# B&R Automation Studio project NAINV104C00R8L515F00 (part 30)

#### Local.var
```iecst
(*2020-09-10*)
(**)
(*Local Action, State & Status*)
VAR
	eAct : eHermesAction := HermesActIdle;
	eStat : eHermesAction := HermesActIdle;
	eMainStatus : eFBStatus := Idle;
	eStatus : eFBStatus := Idle;
	eStatus1 : eFBStatus := Idle;
	eStatus2 : eFBStatus := Idle;
	eStatus3 : eFBStatus := Idle;
	udiStatus : UDINT := 0;
	udiStatus1 : UDINT := 0;
	udiStatus2 : UDINT := 0;
	udiStatus3 : UDINT := 0;
	udiStatus4 : UDINT := 0;
	sStatTxt : STRING[200] := '';
	a_sStatText : ARRAY[0..50] OF STRING[200] := ['Idling','Background Starting Operations','Background Stopping Operations','Deleting Old Log File','Creating Directory','Writing Retain File','Reading Retain File','Saving Configuration',43('')];
END_VAR
(**)
(*Local Alarm*)
VAR
	tyAlmData : tyAlmDat;
	tyAlmData1 : tyAlmDat;
	tyAlmData2 : tyAlmDat;
	tyAlmData3 : tyAlmDat;
	tyAlmData4 : tyAlmDat;
	tyInfoData : tyAlmDat;
	a_tyAlmText : ARRAY[10000..10199] OF tyAlmTxt := [(sAlmText:='Invalid Ident While Creating Server',sRcyText:='Problem Occurred In The TCP/IP Connection. Check The Connection And Try To Reconnect.'),(sAlmText:='Setting Keep Alive Interval Time Error While Creating Server',sRcyText:='Unable To Establish Connection Between Machine. Check For Setting And Resume Operation.'),(sAlmText:='Setting Keep Alive Idle Time Error While Creating Server',sRcyText:='Unable To Establish Connection Between Machine. Check For Setting And Resume Operation.'),(sAlmText:='Setting Keep Alive Count Error While Creating Server',sRcyText:='Unable To Establish Connection Between Machine. Check For Setting And Resume Operation.'),(sAlmText:='Setting Keep Alive Error While Creating Server',sRcyText:='Unable To Establish Connection Between Machine. Check For Setting And Resume Operation.'),(sAlmText:='Setting Receive Buffer Error While Creating Server',sRcyText:='Unable To Establish Connection Between Machine. Check For Setting And Resume Operation.'),(sAlmText:='Setting Send Buffer Error While Creating Server',sRcyText:='Unable To Establish Connection Between Machine. Check For Setting And Resume Operation.'),(sAlmText:='Setting No Waiting Error While Creating Server',sRcyText:='Unable To Establish Connection Between Machine. Check For Setting And Resume Operation.'),(sAlmText:='TCP Open Port Error While Creating Server',sRcyText:='Problem Occurred In The TCP/IP Connection. Check The Connection And Try To Reconnect.'),(sAlmText:='Closing TCP Error While Creating Server',sRcyText:='Problem Occurred In The TCP/IP Connection. Check The Connection And Try To Reconnect.'),(sAlmText:='Invalid Ident While Listening Client',sRcyText:='There Was A Problem Connecting To The Server. The Server May Not Exist or It is Unavailable At This Time. Check The Connection and Try Again.'),(0),(sAlmText:='DS Hermes Connection Lost',sRcyText:='There Was A Problem Connecting To The Server. The Server May Not Exist or It is Unavailable At This Time. Check The Connection and Try Again.'),(0),(sAlmText:='Invalid Ident While Receiving Data',sRcyText:='Problem Occurred In The TCP/IP Connection. Check The Connection And Try To Reconnect.'),(sAlmText:='TCP Receive Data Error While Receiving Data',sRcyText:='Problem Occurred In The TCP/IP Connection. Check The Connection And Try To Reconnect.'),(sAlmText:='Receive BoardAvailable While Downstream In Not Connected State',sRcyText:='Receive Illegal Message.'),(sAlmText:='Receive RevokeBoardAvailable While Downstream In Not Connected State',sRcyText:='Receive Illegal Message.'),(sAlmText:='Receive MachineReady While Downstream In Not Connected State',sRcyText:='Receive Illegal Message.'),(sAlmText:='Receive RevokeMachineReady While Downstream In Not Connected State',sRcyText:='Receive Illegal Message.'),(sAlmText:='Receive StartTransport While Downstream In Not Connected State',sRcyText:='Receive Illegal Message.'),(sAlmText:='Receive StopTransport While Downstream In Not Connected State',sRcyText:='Receive Illegal Message.'),(sAlmText:='Receive TransportFinished While Downstream In Not Connected State',sRcyText:='Receive Illegal Message.'),(sAlmText:='Receive BoardForecast While Downstream In Not Connected State',sRcyText:='Receive Illegal Message.'),(sAlmText:='Receive ServiceDescription While Downstream In Service Description State',sRcyText:='Receive Illegal Message.'),(sAlmText:='Receive BoardAvailable While Downstream In Service Description State',sRcyText:='Receive Illegal Message.'),(sAlmText:='Receive RevokeBoardAvailable While Downstream In Service Description State',sRcyText:='Receive Illegal Message.'),(sAlmText:='Receive MachineReady While Downstream In Service Description State',sRcyText:='Receive Illegal Message.'),(sAlmText:='Receive RevokeMachineReady While Downstream In Service Description State',sRcyText:='Receive Illegal Message.'),(sAlmText:='Receive StartTransport While Downstream In Service Description State',sRcyText:='Receive Illegal Message.'),(sAlmText:='Receive StopTransport While Downstream In Service Description State',sRcyText:='Receive Illegal Message.'),(sAlmText:='Receive TransportFinished While Downstream In Service Description State',sRcyText:='Receive Illegal Message.'),(sAlmText:='Receive BoardForecast While Downstream In Service Description State',sRcyText:='Receive Illegal Message.'),(sAlmText:='Receive ServiceDescription While Downstream In Not Available Not Ready State',sRcyText:='Receive Illegal Message.'),(sAlmText:='Receive BoardAvailable While Downstream In Not Available Not Ready State',sRcyText:='Receive Illegal Message.'),(sAlmText:='Receive RevokeBoardAvailable While Downstream In Not Available Not Ready State',sRcyText:='Receive Illegal Message.'),(sAlmText:='Receive RevokeMachineReady While Downstream In Not Available Not Ready State',sRcyText:='Receive Illegal Message.'),(sAlmText:='Receive StartTransport While Downstream In Not Available Not Ready State',sRcyText:='Receive Illegal Message.'),(sAlmText:='Receive StopTransport While Downstream In Not Available Not Ready State',sRcyText:='Receive Illegal Message.'),(sAlmText:='Receive TransportFinished While Downstream In Not Available Not Ready State',sRcyText:='Receive Illegal Message.'),(sAlmText:='Receive BoardForecast While Downstream In Not Available Not Ready State',sRcyText:='Receive Illegal Message.'),(sAlmText:='Receive ServiceDescription While Downstream In Board Available State',sRcyText:='Receive Illegal Message.'),(sAlmText:='Receive BoardAvailable While Downstream In Board Available State',sRcyText:='Receive Illegal Message.'),(sAlmText:='Receive RevokeBoardAvailable While Downstream In Board Available State',sRcyText:='Receive Illegal Message.'),(sAlmText:='Receive RevokeMachineReady While Downstream In Board Available State',sRcyText:='Receive Illegal Message.'),(sAlmText:='Receive StartTransport While Downstream In Board Available State',sRcyText:='Receive Illegal Message.'),(sAlmText:='Receive StopTransport While Downstream In Board Available State',sRcyText:='Receive Illegal Message.'),(sAlmText:='Receive TransportFinished While Downstream In Board Available State',sRcyText:='Receive Illegal Message.'),(sAlmText:='Receive BoardForecast While Downstream In Board Available State',sRcyText:='Receive Illegal Message.'),(sAlmText:='Receive ServiceDescription While Downstream In Machine Ready State',sRcyText:='Receive Illegal Message.'),(sAlmText:='Receive BoardAvailable While Downstream In Machine Ready State',sRcyText:='Receive Illegal Message.'),(sAlmText:='Receive RevokeBoardAvailable While Downstream In Machine Ready State',sRcyText:='Receive Illegal Message.'),(sAlmText:='Receive MachineReady While Downstream In Machine Ready State',sRcyText:='Receive Illegal Message.'),(sAlmText:='Receive StopTransport While Downstream In Machine Ready State',sRcyText:='Receive Illegal Message.'),(sAlmText:='Receive TransportFinished While Downstream In Machine Ready State',sRcyText:='Receive Illegal Message.'),(sAlmText:='Receive BoardForecast While Downstream In Machine Ready State',sRcyText:='Receive Illegal Message.'),(sAlmText:='Receive ServiceDescription While Downstream In Available And Ready State',sRcyText:='Receive Illegal Message.'),(sAlmText:='Receive BoardAvailable While Downstream In Available And Ready State',sRcyText:='Receive Illegal Message.'),(sAlmText:='Receive RevokeBoardAvailable While Downstream In Available And Ready State',sRcyText:='Receive Illegal Message.'),(sAlmText:='Receive MachineReady While Downstream In Available And Ready State',sRcyText:='Receive Illegal Message.'),(sAlmText:='Receive StopTransport While Downstream In Available And Ready State',sRcyText:='Receive Illegal Message.'),(sAlmText:='Receive TransportFinished While Downstream In Available And Ready State',sRcyText:='Receive Illegal Message.'),(sAlmText:='Receive BoardForecast While Downstream In Available And Ready State',sRcyText:='Receive Illegal Message.'),(sAlmText:='Receive ServiceDescription While Downstream In Transporting State',sRcyText:='Receive Illegal Message.'),(sAlmText:='Receive BoardAvailable While Downstream In Transporting State',sRcyText:='Receive Illegal Message.'),(sAlmText:='Receive RevokeBoardAvailable While Downstream In Transporting State',sRcyText:='Receive Illegal Message.'),(sAlmText:='Receive MachineReady While Downstream In Transporting State',sRcyText:='Receive Illegal Message.'),(sAlmText:='Receive RevokeMachineReady While Downstream In Transporting State',sRcyText:='Receive Illegal Message.'),(sAlmText:='Receive StartTransport While Downstream In Transporting State',sRcyText:='Receive Illegal Message.'),(sAlmText:='Receive TransportFinished While Downstream In Transporting State',sRcyText:='Receive Illegal Message.'),(sAlmText:='Receive BoardForecast While Downstream In Transporting State',sRcyText:='Receive Illegal Message.'),(sAlmText:='Receive ServiceDescription While In Transport Finished State',sRcyText:='Receive Illegal Message.'),(sAlmText:='Receive BoardAvailable While In Transport Finished State',sRcyText:='Receive Illegal Message.'),(sAlmText:='Receive RevokeBoardAvailable While In Transport Finished State',sRcyText:='Receive Illegal Message.'),(sAlmText:='Receive MachineReady While In Transport Finished State',sRcyText:='Receive Illegal Message.'),(sAlmText:='Receive RevokeMachineReady While In Transport Finished State',sRcyText:='Receive Illegal Message.'),(sAlmText:='Receive StartTransport While In Transport Finished State',sRcyText:='Receive Illegal Message.'),(sAlmText:='Receive TransportFinished While In Transport Finished State',sRcyText:='Receive Illegal Message.'),(sAlmText:='Receive BoardForecast While In Transport Finished State',sRcyText:='Receive Illegal Message.'),(sAlmText:='Receive ServiceDescription While Downstream In Transport Stopped State',sRcyText:='Receive Illegal Message.'),(sAlmText:='Receive BoardAvailable While Downstream In Transport Stopped State',sRcyText:='Receive Illegal Message.'),(sAlmText:='Receive RevokeBoardAvailable While Downstream In Transport Stopped State',sRcyText:='Receive Illegal Message.'),(sAlmText:='Receive MachineReady While Downstream In Transport Stopped State',sRcyText:='Receive Illegal Message.'),(sAlmText:='Receive RevokeMachineReady While Downstream In Transport Stopped State',sRcyText:='Receive Illegal Message.'),(sAlmText:='Receive StartTransport While Downstream In Transport Stopped State',sRcyText:='Receive Illegal Message.'),(sAlmText:='Receive StopTransport While Downstream In Transport Stopped State',sRcyText:='Receive Illegal Message.'),(sAlmText:='LaneId Mismatch While Checking Service Description',sRcyText:='The LaneId Value Does Not Match. Change The Value And Resend The Value.'),(sAlmText:='MachineId Missing While Checking Service Description',sRcyText:='Missing Input Value For MachineId. Fill Up The Value And Resend.'),(sAlmText:='LandId Out Of Range While Checking Service Description',sRcyText:='LaneId Does Not Fall Within The Expected Range.'),(sAlmText:='LandId Missing While Checking Service Description',sRcyText:='Missing Input Value For LaneId. Fill Up The Value And Resend.'),(sAlmText:='Version Missing While Checking Service Description',sRcyText:='Missing Input Value For Version. Fill Up The Value And Resend.'),(sAlmText:='SupportedFeatures Missing While Checking Service Description',sRcyText:='Missing Input Value For SupportedFeatures. Fill Up The Value And Resend.'),(sAlmText:='NotificationCode Out Of Range While Checking Notification',sRcyText:='NotificationCode Does Not Fall Within The Expected Range.'),(sAlmText:='NotificationCode Missing While Checking Notification',sRcyText:='Missing Input Value For NotificationCode. Fill Up The Value And Resend.'),(sAlmText:='Severity Missing While Checking Notification',sRcyText:='Missing Input Value For Severity. Fill Up The Value And Resend.'),(sAlmText:='Description Missing While Checking Notification',sRcyText:='Missing Input Value For Description. Fill Up The Value And Resend.'),2((0)),(sAlmText:='FailedBoard Missing While Checking Machine Ready',sRcyText:='Missing Input Value For FailedBoard. Fill Up The Value And Resend.'),(sAlmText:='TransferState Missing While Checking Stop Transport',sRcyText:='Missing Input Value For TransferState. Fill Up The Value And Resend.'),(sAlmText:='BoardId Missing While Checking Stop Transport',sRcyText:='Missing Input Value For BoardId. Fill Up The Value And Resend.'),(sAlmText:='BoardId Missing While Checking Start Transport',sRcyText:='Missing Input Value For BoardId. Fill Up The Value And Resend.'),(sAlmText:='Barcode Missing While Checking Query Board Info',sRcyText:='Missing Input Value For BoardId. Fill Up The Value And Resend.'),(0),(sAlmText:='BoardId Mismatch While Checking Start Transport & Stop Transport',sRcyText:='The BoardId Value Does Not Match. Change The Value And Resend The Value.'),(sAlmText:='BoardId Missing While Checking Start Transport & Stop Transport',sRcyText:='Missing Input Value For BoardId. Fill Up The Value And Resend.'),(sAlmText:='Service Description Interchange Time Out',sRcyText:='Timeout Expired Before Operation Completed. Reset And Resume Operation.'),(sAlmText:='Transport Time Out',sRcyText:='Timeout Expired Before Operation Completed. Reset And Resume Operation.'),(sAlmText:='Receive TransportFinished While Downstream In Transport Stopped State',sRcyText:='Receive Illegal Message.'),(sAlmText:='Receive BoardForecast While Downstream In Transport Stopped State',sRcyText:='Receive Illegal Message.'),(sAlmText:='Stop Transport Request To Send From Upstream Hermes',sRcyText:='Sending Illegal Message.'),(sAlmText:='Get Directory Info Error While Deleting Old Log',sRcyText:='An Error Was Encountered While Getting Directory Info. Please Contact Nutek For A Possible Solution.'),(sAlmText:='Directory Read Error While Deleting Old Log',sRcyText:='An Error Was Encountered While Reading Directory. Please Contact Nutek For A Possible Solution.'),(sAlmText:='File Delete Error While Deleting Old Log',sRcyText:='An Error Was Encountered While Trying To Delete File. Please Contact Nutek For A Possible Solution.'),18((0)),(sAlmText:='Check Alive Time Out',sRcyText:='Timeout Expired Before Operation Completed. Reset And Resume Operation.'),(sAlmText:='Waiting Check Alive Time Out',sRcyText:='Timeout Expired Before Operation Completed. Reset And Resume Operation.'),(sAlmText:='Check Alive Id Mismatch',sRcyText:='The Check Alive Id Value Does Not Match. Change The Value And Resend The Value.'),(sAlmText:='Machine Ready Request To Send From Upstream Hermes',sRcyText:='Sending Illegal Message.'),(sAlmText:='Revoke Machine Ready Request To Send From Upstream Hermes',sRcyText:='Sending Illegal Message.'),(sAlmText:='Start Transport Request To Send From Upstream Hermes',sRcyText:='Sending Illegal Message.'),(sAlmText:='Set Configuration Request To Send From Upstream Hermes',sRcyText:='Sending Illegal Message.'),(sAlmText:='Get Configuration Request To Send From Upstream Hermes',sRcyText:='Sending Illegal Message.'),(sAlmText:='Current Configuration Request To Send From Upstream Hermes',sRcyText:='Sending Illegal Message.'),(sAlmText:='Board Forecast Request To Send From Upstream Hermes',sRcyText:='Sending Illegal Message.'),(sAlmText:='Query Board Info Request To Send From Upstream Hermes',sRcyText:='Sending Illegal Message.'),(sAlmText:='Invalid Ident While Sending Data',sRcyText:='Invalid Ident Value.'),(sAlmText:='TCP Retry Send Data Error While Sending Data',sRcyText:='Problem Occurred In The TCP/IP Connection. Check The Connection And Try To Reconnect.'),(sAlmText:='TCP Send Data Error',sRcyText:='Problem Occurred In The TCP/IP Connection. Check The Connection And Try To Reconnect.'),(sAlmText:='Invalid Ident While Closing TCP',sRcyText:='Invalid Ident Value.'),(sAlmText:='Closing TCP Error',sRcyText:='Problem Occurred In The TCP/IP Connection. Check The Connection And Try To Reconnect.'),(sAlmText:='File Open Error While Writing Log',sRcyText:='An Error Was Encountered While Trying To Open File. Please Contact Nutek For A Possible Solution.'),(sAlmText:='File Create Error While Writing Log',sRcyText:='An Error Was Encountered While Trying To Create File. Please Contact Nutek For A Possible Solution.'),(sAlmText:='Get File Info Error While Writing Log',sRcyText:='An Error Was Encountered While Getting File Info. Please Contact Nutek For A Possible Solution.'),(sAlmText:='File Write Error While Writing Log',sRcyText:='An Error Was Encountered While Trying To Write File. Please Contact Nutek For A Possible Solution.'),(sAlmText:='File Close Error While Writing Log',sRcyText:='An Error Was Encountered While Trying To Close File. Please Contact Nutek For A Possible Solution.'),(sAlmText:='Directory Does Not Exist While Writing Log',sRcyText:='The Directory Does Not Exist.Please Contact Nutek For A Possible Solution.'),(sAlmText:='Invalid Ident While Closing TCP',sRcyText:='Invalid Ident Value.'),(sAlmText:='Closing TCP Error',sRcyText:='Problem Occurred In The TCP/IP Connection. Check The Connection And Try To Reconnect.'),(0),(sAlmText:='Board Jam At Sensor After Transfer Interrupted',sRcyText:='Pull Back Board From Downstream Machine'),42((0))];
END_VAR
(**)
(*Local Output*)
VAR
	bConnected : BOOL;
	bHandshakeDone : BOOL;
	bUSRdy : BOOL;
	bDSRdy : BOOL;
	bUSGdRdy : BOOL;
	bDSGdRdy : BOOL;
	bTransporting : BOOL;
	bStopTransport : BOOL;
	sInternalSnd : STRING[65535];
END_VAR
(**)
(*Local Input*)
VAR
	udiRstErr : UDINT := 0;
	bPrep : BOOL := TRUE;
	bEn : BOOL := TRUE;
	bDis : BOOL := FALSE;
	tyParam : tyHermesDSParam;
	sIPAddr : STRING[15] := '192.168.0.100';
	a_usiMacAddr : ARRAY[0..5] OF USINT := [6(0)];
	tyDTStructure : DTStructure := (year:=2019,month:=01,day:=05,wday:=05,hour:=21,minute:=28,second:=30,millisec:=123,microsec:=456);
	dtCurrDT : DATE_AND_TIME := DT#2019-02-23-12:30:50;
	bRdySnd : BOOL := FALSE;
	bSndCompl : BOOL := FALSE;
	bSndInCompl : BOOL := FALSE;
	bSndNotStart : BOOL := FALSE;
	bBAWidthEn : BOOL := TRUE; (*Board Available Check Width*)
	bBASltEn : BOOL := FALSE; (*Board Available Check Slot*)
	bBFWidthEn : BOOL := TRUE; (*Board Available Check Width*)
	bBFSltEn : BOOL := FALSE; (*Board Available Check Slot*)
	sMcId : STRING[80] := '';
	sInterfaceId : STRING[80];
	sVersion : STRING[7] := '1.0.2';
	eFailedBoard : eHermesFailedBoard := HermesUnknownBoard;
	sRecipeNm : STRING[254] := '';
	eFlippedBoard : eHermesFlippedBoard := HermesFlippedBoardUnknownSide;
	sTopBarcode : STRING[254] := '';
	sBottomBarcode : STRING[254] := '';
	rLength : REAL := 0;
	rThickness : REAL := 0;
	rConveyorSpeed : REAL := 0;
	rTopClearanceHeight : REAL := 0;
	rBottomClearanceHeight : REAL := 0;
	rWeight : REAL := 0;
	sWorkOrderId : STRING[80] := '';
	sBatchId : STRING[80] := '';
	diWidthInUM : DINT := 0;
	diMinSltValue : DINT := 0;
	diMaxSltValue : DINT := 0;
	diPitch : DINT := 0;
	diTtlSlt : DINT := 0;
	diSltToSltInUM : DINT := 0;
	udiSndBffrSize : UDINT := 65536;
	udiRcvBffrSize : UDINT := 65536;
	udiAliveIdleTimeInSec : UDINT := 5;
	tConnTimeOut : TIME := T#30s;
	diTransferInTO : DINT := 30000;
	a_tyXMLTableDataBrdAvl : ARRAY[0..200] OF tyXMLTableDat;
	iXMLTableDataBrdAvlTtlIdx : INT := 0;
	bNewBrdAvl : BOOL := FALSE;
	bOpsRun : BOOL := FALSE;
	bInterruptSen : BOOL := FALSE;
	udiFileKeepDay : UDINT := 30;
	sProgNm : STRING[15] := 'DSHermes';
	bNtSettingsLoadDone : BOOL := TRUE;
	sRmtMcId : STRING[80];
	bRmtPrep : BOOL := FALSE;
	bRmtEn : BOOL := FALSE;
	bInternalUse : BOOL;
	sInternalRcv : STRING[65535];
END_VAR
(**)
(*Local*)
VAR
	bRstErr : BOOL;
	udiRstErrOld : UDINT;
	bInitDone : BOOL;
	bInitialDone : BOOL;
	bRun : BOOL;
	bStop : BOOL;
	bRstConnection : BOOL;
	bRstState : BOOL;
	udiSvrIdent : UDINT;
	udiClntIdent : UDINT;
	udiClntIdentExtra : UDINT;
	udiXMLTableWriteIdx : UDINT;
	udiMsgSendBffr : UDINT;
	udiMsgCmdBffr : UDINT;
	udiSndMsgLen : UDINT;
	sSnd : STRING[65535];
	sRcv : STRING[65535];
	a_tyXMLTableDataRcv : ARRAY[0..200] OF tyXMLTableDat;
	a_tyXMLTableDataSnd : ARRAY[0..200] OF tyXMLTableDat;
	a_eMsgSend : ARRAY[0..50] OF eHermesMsgType;
	a_eCommandSndQ : ARRAY[0..20] OF eHermesCommand;
	tyMsgTypeRcv : tyHermesMsgType;
	tyCheckAliveSnd : tyHermesCheckAlive;
	tyCheckAlivePingSnd : tyHermesCheckAlive;
	tyCheckAlivePongSnd : tyHermesCheckAlive;
	tyCheckAliveRcv : tyHermesCheckAlive;
	tyCheckAlivePingRcv : tyHermesCheckAlive;
	tyCheckAlivePongRcv : tyHermesCheckAlive;
	tyServiceDescriptionSnd : tyHermesServiceDescription;
	tyServiceDescriptionRcv : tyHermesServiceDescription;
	tyNotificationSnd : tyHermesNotification;
	tyNotificationRcv : tyHermesNotification;
	tyBoardAvailableRcv : tyHermesBoardAvailable;
	tyBoardAvailableSnd : tyHermesBoardAvailable;
	a_tyBoardDepartedInfo : ARRAY[0..49] OF tyHermesBoardAvailable;
	a_tyBoardDepartedInfoWr : ARRAY[0..49] OF tyHermesBoardAvailable;
	tyMachineReady : tyHermesMachineReady;
	tyStartTransport : tyHermesStartTransport;
	tyStopTransport : tyHermesStopTransport;
	tyTransportFinished : tyHermesTransportFinished;
	tySetConfiguration : tyHermesSetConfiguration;
	tyCurrentConfiguration : tyHermesCurrentConfiguration;
	tyBoardForecastRcv : tyHermesBoardForecast;
	tyBoardForecastSnd : tyHermesBoardForecast;
	tyQueryBoardInfo : tyHermesQueryBoardInfo;
	tySendBoardInfo : tyHermesSendBoardInfo;
	tyCommandRcv : tyHermesCommand;
	tyCommandSnd : tyHermesCommand;
	fbCreateSvr : fbTCPCreateSvr;
	fbListen : fbTCPListen;
	fbRcv : fbTCPRcv;
	fbSend : fbTCPSnd;
	fbCloseSvr : fbTCPClose;
	fbCloseClnt : fbTCPClose;
	fbParseXMLTable : fbHermesParseXMLTable;
	fbParseBrdAvlExternal : fbHermesParseXMLTable;
	fbCheckAlive : fbHermesCheckAlive;
	fbCheckAliveSendPing : fbHermesCheckAliveSendPing;
	fbCheckAliveRcvPing : fbHermesCheckAliveRcvPing;
	fbSequenceDS : fbHermesSequenceDS;
	fbSequenceTO : fbHermesSequenceTO;
END_VAR
VAR RETAIN
	usiBAIndex : USINT := 0;
END_VAR
VAR
	usiPrevBAIndex : USINT;
	eStatOld : eHermesAction := HermesActIdle;
	tyParamOld : tyHermesDSParam;
	udiLogCntr : UDINT := 1;
	udiWriteLogCntr : UDINT := 1;
	a_sLogList : ARRAY[1..10] OF STRING[65535];
	sDT : STRING[80];
	dtCurrDTTemp : DATE_AND_TIME;
	fbFileAppend1 : fbFileFullAppend;
	fbFileOldDel1 : fbFileOldDel;
	fbFileRead1 : fbFileFullRead;
	fbFileWrite1 : fbFileFullWrite;
	iWriteLogStep : INT := 0;
	tyUSHermestyBoardAvailable : tyHermesBoardAvailable;
	tyCommandParam : tyHermesCommandParam;
	bDummy : BOOL;
	bFeatureBoardForecast : BOOL;
	bNewProduct : BOOL;
	bNewWidth : BOOL;
	bNewChangeOver : BOOL;
	tySendBoardInfoAcc : tyHermesSendBoardInfo;
	rMachineCycleTime : REAL;
	rAWCycleTm : REAL;
	bFileNotFound : BOOL;
	bSendBFId : BOOL;
	bBFIdSent : BOOL;
	bSendBFNoID : BOOL;
	bSndReverseBF : BOOL;
	bRstSendBFId : BOOL;
	bFirstZoneHaveBoard : BOOL;
	bFirstZoneEndSen : BOOL;
	bAllZoneEmpty : BOOL;
	bTransportFinishedSnd : BOOL;
	fbTimerRstBFId : TON;
	sInfoMcRdyMsg : STRING[200];
	sTempRealWidth : STRING[15];
	sRstTim : STRING[15];
	udiModuleNum : UDINT := 3351;
END_VAR
(*Send Board Info*)
VAR
	bSearchTop : BOOL;
	bSearchBottom : BOOL;
	siTopBarcodeIdx : SINT;
	siBottomBarcodeIdx : SINT;
	siSearhIdx : SINT;
	siFoundIdx : SINT;
	bCompleteSearch : BOOL;
END_VAR
(*Route*)
VAR
	bTriggerRouteReversal : BOOL;
	bReverseDSSndBfWBrdID : BOOL;
	bSwitchtoReverseSend : BOOL;
	fbRstReverseSndGate : TON;
	bNotifyRstReverseSndGate : BOOL;
	bBlkDS : BOOL;
	bProcessRouteEn : BOOL;
	bManualRmvRoute : BOOL;
	bReturnRoute : BOOL;
	bNomRouteEn : BOOL;
	bReverseSentRoute : BOOL;
	usiUSHermesReverseDSSendBFId : USINT;
	bUSHermesProcessRouteTrigger : BOOL;
	iRoute : INT;
	iAction : INT;
	bDSHermesRcvReverseUSMcRdy : BOOL;
	bReverseRcvBlkDS : BOOL;
END_VAR
```

#### Act_Action.st
```iecst
(** 2021-08-01 **)
ACTION Act_Action:

	//Reset Error
	IF (eStatus = Error) AND bRstErr THEN
		p_eAct	:= HermesActIdle;
		eStat	:= HermesActIdle;
	END_IF

	//Set p_eAct
	IF eStatus = Idle  OR eStatus = Done THEN //OR eStatus = Busy
		eStat	:= p_eAct;
	END_IF

END_ACTION
```

#### Act_Alarm.st
```iecst
(** 2021-08-01 **)
ACTION Act_Alarm:

	//Error
	IF EDGEPOS(eStatus = Error) THEN

		tyAlmData.sProgNm		:= p_sProgNm;
		tyAlmData.udiCode		:= udiStatus;
		tyAlmData.eSeverity		:= AlmSeverityError;
		tyAlmData.udiRunTime	:= tyAlmData.udiRunTime + 1;
		tyAlmData.bAlm			:= TRUE;
		tyAlmData.udiModuleNum  := udiModuleNum;
		g_sDSHermesProgNm		:= p_sProgNm;

		//Get Error Message
		IF tyAlmData.udiCode < 10000 OR tyAlmData.udiCode > 10199 THEN
			tyAlmData.sAlmMsg	:= 'Unknown';
			tyAlmData.sRcyMsg	:= 'Unknown';
		ELSE
			tyAlmData.sAlmMsg	:= a_tyAlmText[tyAlmData.udiCode].sAlmText;
			tyAlmData.sRcyMsg	:= a_tyAlmText[tyAlmData.udiCode].sRcyText;
		END_IF

		sStatTxt	:= tyAlmData.sAlmMsg;

	ELSIF bRstErr AND (tyAlmData.udiCode <> 0) THEN

		tyAlmData.udiCode	:= 0;
		tyAlmData.eSeverity	:= AlmSeverityNA;
		tyAlmData.sAlmMsg	:= '';
		tyAlmData.sRcyMsg	:= '';
		tyAlmData.bAlm			:= FALSE;
		sStatTxt	:= a_sStatText[eStat];

	END_IF

END_ACTION
```

#### Act_Alarm1.st
```iecst
(** 2021-08-01 **)
ACTION Act_Alarm1: //General

	//Error
	IF EDGEPOS(eStatus1 = Error) THEN

		tyAlmData1.sProgNm		:= p_sProgNm;
		tyAlmData1.udiCode		:= udiStatus1;
		tyAlmData1.eSeverity	:= AlmSeverityError;
		tyAlmData1.udiRunTime	:= tyAlmData1.udiRunTime + 1;
		tyAlmData1.bAlm			:= TRUE;
		tyAlmData1.udiModuleNum := udiModuleNum;
		g_sDSHermesProgNm		:= p_sProgNm;

		//Get Error Message
		IF tyAlmData1.udiCode < 10000 OR tyAlmData1.udiCode > 10199 THEN
			tyAlmData1.sAlmMsg	:= 'Unknown';
			tyAlmData1.sRcyMsg	:= 'Unknown';
		ELSE
			tyAlmData1.sAlmMsg	:= a_tyAlmText[tyAlmData1.udiCode].sAlmText;
			tyAlmData1.sRcyMsg	:= a_tyAlmText[tyAlmData1.udiCode].sRcyText;
		END_IF

		sStatTxt	:= tyAlmData1.sAlmMsg;

	ELSIF bRstErr AND (tyAlmData1.udiCode <> 0) THEN

		tyAlmData1.udiCode		:= 0;
		tyAlmData1.eSeverity	:= AlmSeverityNA;
		tyAlmData1.sAlmMsg		:= '';
		tyAlmData1.sRcyMsg		:= '';
		tyAlmData1.bAlm			:= FALSE;
		sStatTxt	:= a_sStatText[eStat];

	END_IF

END_ACTION
```

#### Act_Background_BoardForecast.st
```iecst
(** 2023-08-01 **)
ACTION Act_Background_BoardForecast:

//	bSndReverseBF := p_bUSHermesReverseDSSendBFId

	bFeatureBoardForecast := (p_tyParam.bFeatureBoardForecast = TRUE) AND (tyServiceDescriptionRcv.tyAvl.tySupportedFeatures.bFeatureBoardForecast = TRUE) (*AND bHandshakeDone*) ;

	IF NOT(bFeatureBoardForecast) THEN
		bNewChangeOver := FALSE;
		bSendBFNoID	   := FALSE;
		bSendBFId	   := FALSE;
		bBFIdSent	   := FALSE;
		bSndReverseBF  :=  FALSE;
		tyInfoData.sProgNm		:= '';
		tyInfoData.udiCode		:= 0;
		tyInfoData.eSeverity	:= AlmSeverityNA;
		tyInfoData.sAlmMsg		:= '';
	ELSE
		bSndReverseBF := EDGEPOS(p_usiUSHermesReverseDSSendBFId <> 0);

		fbTimerRstBFId(IN:= bSendBFId AND bBFIdSent
		AND NOT(bRstSendBFId) AND tyInfoData.udiCode= 10999
		AND bDSRdy
		,PT := T#1000s); //start counting when received mismatch Machine ready

		IF bRstSendBFId OR fbTimerRstBFId.Q
			OR EDGEPOS(bAllZoneEmpty AND p_bConvInitDone)  THEN //Reset BoardForecast width id
			bRstSendBFId := FALSE;
			bSendBFId := FALSE;
			bBFIdSent := FALSE;
		ELSIF fbTimerRstBFId.IN THEN
			sRstTim 				:= REAL_TO_STRING(TIME_TO_REAL(fbTimerRstBFId.PT-fbTimerRstBFId.ET)/1000.0);
			tyInfoData.sAlmMsg		:= CONCAT(sInfoMcRdyMsg,CONCAT(sRstTim,'(seconds)'));
		END_IF

		IF EDGEPOS(bNewProduct) OR EDGEPOS(bNewWidth) THEN  //Trigger BFID
			bNewChangeOver := TRUE;
			bBFIdSent := FALSE; //To resend BF-ID
		END_IF

		IF bNewChangeOver AND bAllZoneEmpty AND p_bConvInitDone THEN
			bNewChangeOver:= FALSE;
			bSendBFId	  := TRUE; //reset when find mactch machine ready
		END_IF

		IF bSendBFId = FALSE AND bBFIdSent = FALSE THEN //reset notification
			tyInfoData.sProgNm		:= '';
			tyInfoData.udiCode		:= 0;
			tyInfoData.eSeverity	:= AlmSeverityNA;
			tyInfoData.sAlmMsg		:= '';
		END_IF

		IF bSendBFId = FALSE   THEN  	//Trigger BF No Id
			bSendBFNoID	:= FALSE;
			IF bFirstZoneHaveBoard AND NOT(bFirstZoneEndSen) THEN //Zone 1 PCB_In and have Board
				bSendBFNoID	:= TRUE;
			ELSIF bSndReverseBF THEN//EDGEPOS(bSndReverseBF) OR EDGENEG(bSndReverseBF) THEN //Reverse route
				bSendBFNoID	:= TRUE; //EDGEPOS send Brd id , EDGENEG send empty brd id
			END_IF
		END_IF

	END_IF

END_ACTION
```

#### Act_Background_ChgConfig.st
```iecst
(** 2021-08-01 **)
ACTION Act_Background_ChgConfig:

	IF eStatus2 <> Error THEN

		IF (tyParamOld.iLaneID <> p_tyParam.iLaneID) OR (tyParamOld.sClientAddress <> p_tyParam.sClientAddress) OR (tyParamOld.uiClientPort <> p_tyParam.uiClientPort) OR (tyParamOld.uiSvrPort <> p_tyParam.uiSvrPort)
			OR (tyParamOld.bFeatureBoardForecast <> p_tyParam.bFeatureBoardForecast) OR (tyParamOld.bFeatureCheckAliveResponse <> p_tyParam.bFeatureCheckAliveResponse) OR (tyParamOld.bFeatureSendBoardInfo <> p_tyParam.bFeatureSendBoardInfo) THEN

			IF udiClntIdent <> 0 THEN
				fHermesAddOneMsgSend(ADR(a_eMsgSend) , ADR(udiMsgSendBffr) , HermesMsgTypeNotification);

				tyNotificationSnd.tyAvl.bSeverity			:= TRUE;
				tyNotificationSnd.tyAvl.bNotificationCode	:= TRUE;
				tyNotificationSnd.tyAvl.bDescription		:= TRUE;
				tyNotificationSnd.tyData.eSeverity			:= HermesSeverityFatalError;
				tyNotificationSnd.tyData.iNotificationCode	:= 3;
				tyNotificationSnd.tyData.sDescription		:= 'Configuration Changed';

			END_IF

			bRstConnection	:= TRUE;

		END_IF

	END_IF

END_ACTION
```

#### Act_Background_ChkAlive.st
```iecst
(** 2019-05-30 **)
ACTION Act_Background_ChkAlive:

	IF eStatus1 <> Error THEN

		//Standard Check Alive (Without Ping & Pong)
		fbCheckAlive.bDataRcv		:= tyMsgTypeRcv.bCheckAlive OR tyMsgTypeRcv.bMachineReady OR tyMsgTypeRcv.bRevokeMachineReady OR tyMsgTypeRcv.bStartTransport OR tyMsgTypeRcv.bStopTransport OR tyMsgTypeRcv.bQueryBoardInfo;
		fbCheckAlive.tSendTm		:= p_tyParam.tSndAlive;
		fbCheckAlive.tRcvTimeOut	:= p_tyParam.tRcvAlive;
		fbCheckAlive(bEn := TRUE);

		IF fbCheckAlive.udiStatus > 0 AND fbCheckAlive.udiStatus < 65534 THEN
			eStatus1	:= Error;

			IF fbCheckAlive.udiStatus = 2767 THEN
				udiStatus1	:= 10132;	//Check Alive Time Out
			ELSE
				udiStatus1	:= fbCheckAlive.udiStatus;
			END_IF

			fHermesAddOneMsgSend(ADR(a_eMsgSend) , ADR(udiMsgSendBffr) , HermesMsgTypeNotification);

			tyNotificationSnd.tyAvl.bSeverity			:= TRUE;
			tyNotificationSnd.tyAvl.bNotificationCode	:= TRUE;
			tyNotificationSnd.tyAvl.bDescription		:= TRUE;
			tyNotificationSnd.tyData.eSeverity			:= HermesSeverityFatalError;
			tyNotificationSnd.tyData.iNotificationCode	:= UDINT_TO_INT(udiStatus1);
			tyNotificationSnd.tyData.sDescription		:= a_tyAlmText[udiStatus1].sAlmText;

		ELSE
			IF EDGEPOS(fbCheckAlive.bDataSend) THEN
				fHermesAddOneMsgSend(ADR(a_eMsgSend) , ADR(udiMsgSendBffr) , HermesMsgTypeCheckAlive);
				tyCheckAliveSnd	:= fbCheckAlive.tyDataSend;
			END_IF

		END_IF

		tyMsgTypeRcv.bCheckAlive	:= FALSE;	//Reset Check Alive

	END_IF

END_ACTION
```

#### Act_Background_CmpParamRcv.st
```iecst
(** 2021-08-01 **)
ACTION Act_Background_CmpParamRcv:

	IF eStatus2 <> Error THEN

		IF tyMsgTypeRcv.bStopTransport = TRUE THEN
			udiStatus2	:= fHermesChkParamSTST(tyStartTransport , tyStopTransport);

			IF udiStatus2 <> 0 THEN
				eStatus2	:= Error;

				IF udiStatus2 = 2712 THEN
					udiStatus2	:= 10104;	//BoardId Mismatch While Checking Start Transport & Stop Transport
				ELSIF udiStatus2 = 2713 THEN
					udiStatus2	:= 10105;	//BoardId Missing While Checking Start Transport & Stop Transport
				END_IF

				fHermesAddOneMsgSend(ADR(a_eMsgSend) , ADR(udiMsgSendBffr) , HermesMsgTypeNotification);

				tyNotificationSnd.tyAvl.bSeverity			:= TRUE;
				tyNotificationSnd.tyAvl.bNotificationCode	:= TRUE;
				tyNotificationSnd.tyAvl.bDescription		:= TRUE;
				tyNotificationSnd.tyData.eSeverity			:= HermesSeverityFatalError;
				tyNotificationSnd.tyData.iNotificationCode	:= UDINT_TO_INT(udiStatus2);
				tyNotificationSnd.tyData.sDescription		:= a_tyAlmText[udiStatus2].sAlmText;

			END_IF
		END_IF

		IF tyMsgTypeRcv.bStartTransport = TRUE THEN
			IF fHermesChkParamBAST(tyBoardAvailableSnd , tyStartTransport) <> 0 THEN
				p_bSndNotStart	:= TRUE;
			END_IF
		END_IF

		IF bFeatureBoardForecast THEN	//HermesMsgTypeBoardForecast
			IF fbSequenceDS.eState = HermesStateMachineReady   AND bSendBFId AND bBFIdSent THEN
				udiStatus2	:= fHermesChkParamBFMR(tyBoardForecastSnd , tyMachineReady); //Modify this if our machine need to Error when ForecastId in MachineReady(Id) received is different

				IF udiStatus2 <> 0 THEN //Alarm Info
					memset(ADR(sInfoMcRdyMsg),0,SIZEOF(sInfoMcRdyMsg));
					sInfoMcRdyMsg := CONCAT(sInfoMcRdyMsg , 'Details mismatch between BoardForecast and MachineReady');
					sInfoMcRdyMsg := CONCAT(sInfoMcRdyMsg , '$r$n');
					IF udiStatus2 = 2716 THEN 	//Forecast Id Mismatch While Checking BoardForecast & Machine Ready
						sInfoMcRdyMsg := CONCAT(sInfoMcRdyMsg , 'ForecastID sent:');
						sInfoMcRdyMsg := CONCAT(sInfoMcRdyMsg , tyBoardForecastSnd.tyData.sForecastId);
						sInfoMcRdyMsg := CONCAT(sInfoMcRdyMsg , '$r$n');
						sInfoMcRdyMsg := CONCAT(sInfoMcRdyMsg , 'ForecastID received:');
						sInfoMcRdyMsg := CONCAT(sInfoMcRdyMsg , tyMachineReady.tyData.sForecastId);
					ELSIF udiStatus2 = 2717 THEN 	//Product Type Id Mismatch While Checking BoardForecast & Machine Ready
						sInfoMcRdyMsg := CONCAT(sInfoMcRdyMsg , 'ProductType sent:');
						sInfoMcRdyMsg := CONCAT(sInfoMcRdyMsg , tyBoardForecastSnd.tyData.sProductTypeId);
						sInfoMcRdyMsg := CONCAT(sInfoMcRdyMsg , '$r$n');
						sInfoMcRdyMsg := CONCAT(sInfoMcRdyMsg , 'ProductType received:');
						sInfoMcRdyMsg := CONCAT(sInfoMcRdyMsg , tyMachineReady.tyData.sProductTypeId);
					ELSIF udiStatus2 = 2718 THEN //Width Mismatch While Checking Board Forecast & Machine Ready
						sInfoMcRdyMsg := CONCAT(sInfoMcRdyMsg , 'Width sent:');
						sTempRealWidth := REAL_TO_STRING(tyBoardForecastSnd.tyData.rWidth);
						sInfoMcRdyMsg := CONCAT(sInfoMcRdyMsg ,sTempRealWidth );
						sInfoMcRdyMsg := CONCAT(sInfoMcRdyMsg , '$r$n');
						sInfoMcRdyMsg := CONCAT(sInfoMcRdyMsg , 'Width received:');
						sTempRealWidth := REAL_TO_STRING(tyMachineReady.tyData.rWidth);
						sInfoMcRdyMsg := CONCAT(sInfoMcRdyMsg , sTempRealWidth);
					END_IF
					sInfoMcRdyMsg := CONCAT(sInfoMcRdyMsg , '$r$n');
					sInfoMcRdyMsg := CONCAT(sInfoMcRdyMsg , 'Waiting New MachineReady or Ignore in:');

					tyInfoData.sProgNm		:= p_sProgNm;
					tyInfoData.udiCode		:= 10999;
					tyInfoData.eSeverity	:= AlmSeverityInfo;
					tyInfoData.sAlmMsg		:= sInfoMcRdyMsg;

				ELSE
					bRstSendBFId := TRUE; //Reset bSendBFId if MachineReady(Id) or MachineReady() received is ok
				END_IF

			END_IF
		END_IF

	END_IF

END_ACTION
```

#### Act_Background_Command.st
```iecst
(** 2021-08-01 **)
ACTION Act_Background_Command:
	//tyServiceDescriptionRcv.tyAvl.tySupportedFeatures.bFeatureCommand = TRUE AND p_tyParam.bFeatureCommand AND

	IF NOT(p_tyParam.bFeatureCommand AND tyServiceDescriptionRcv.tyAvl.tySupportedFeatures.bFeatureCommand AND bHandshakeDone) THEN
		IF tyCommandParam.a_eCommandSndQ[0] <> HermesCommandUndefined THEN
			fHermesRmvOneCmdTyp(ADR(tyCommandParam.a_eCommandSndQ),ADR(tyCommandParam.udiMsgCmdBffr));
		END_IF
	ELSE
		IF eStatus2 <> Error THEN
			//receive command

			IF tyMsgTypeRcv.bCommand THEN
				tyCommandParam.usiCommandIdx :=  tyCommandParam.usiCommandIdx + 1;
				tyCommandParam.eCommand := tyCommandRcv.tyData.eCommand;
				tyMsgTypeRcv.bCommand  := FALSE;
			END_IF

			//sending
			IF  tyCommandParam.a_eCommandSndQ[0] <> HermesCommandUndefined THEN
				//Queuing for sending command
				fHermesAddOneMsgSend(ADR(a_eMsgSend) , ADR(udiMsgSendBffr) , HermesMsgTypeCommand);
				tyCommandSnd.tyData.eCommand :=  tyCommandParam.a_eCommandSndQ[0];
				tyCommandSnd.tyAvl.bCommand :=  TRUE;
				fHermesRmvOneCmdTyp(ADR(tyCommandParam.a_eCommandSndQ),ADR(tyCommandParam.udiMsgCmdBffr));
			END_IF
		END_IF
	END_IF

END_ACTION
```

#### Act_Background_Err.st
```iecst
(** 2021-08-01 **)
ACTION Act_Background_Err:

	IF bTransporting = TRUE THEN
		IF bStopTransport AND p_bInterruptSen THEN
			eStatus2	:= Error;
			udiStatus2	:= 10157;	//Board Jam At Sensor After Transfer Interrupted
		END_IF
	END_IF

END_ACTION
```

#### Act_Background_IllegalMsg.st
```iecst
(** 2021-08-01 **)
ACTION Act_Background_IllegalMsg:

	IF eStatus2 <> Error THEN

		udiStatus2	:= fHermesIllegalMsgDS(fbSequenceDS.eState , tyMsgTypeRcv);

		IF udiStatus2 <> 0 THEN
			eStatus2	:= Error;

			IF udiStatus2 = 2840 THEN
				udiStatus2	:= 10016;	//Receive BoardAvailable While Downstream In Not Connected State
			ELSIF udiStatus2 = 2841 THEN
				udiStatus2	:= 10017;	//Receive RevokeBoardAvailable While Downstream In Not Connected State
			ELSIF udiStatus2 = 2842 THEN
				udiStatus2	:= 10018;	//Receive MachineReady While Downstream In Not Connected State
			ELSIF udiStatus2 = 2843 THEN
				udiStatus2	:= 10019;	//Receive RevokeMachineReady While Downstream In Not Connected State
			ELSIF udiStatus2 = 2844 THEN
				udiStatus2	:= 10020;	//Receive StartTransport While Downstream In Not Connected State
			ELSIF udiStatus2 = 2845 THEN
				udiStatus2	:= 10021;	//Receive StopTransport While Downstream In Not Connected State
			ELSIF udiStatus2 = 2846 THEN
				udiStatus2	:= 10022;	//Receive TransportFinished While Downstream In Not Connected State
			ELSIF udiStatus2 = 2847 THEN
				udiStatus2	:= 10023;	//Receive BoardForecast While Downstream In Not Connected State
			ELSIF udiStatus2 = 2848 THEN
				udiStatus2	:= 10024;	//Receive ServiceDescription While Downstream In Service Description State
			ELSIF udiStatus2 = 2849 THEN
				udiStatus2	:= 10025;	//Receive BoardAvailable While Downstream In Service Description State
			ELSIF udiStatus2 = 2850 THEN
				udiStatus2	:= 10026;	//Receive RevokeBoardAvailable While Downstream In Service Description State
			ELSIF udiStatus2 = 2851 THEN
				udiStatus2	:= 10027;	//Receive MachineReady While Downstream In Service Description State
			ELSIF udiStatus2 = 2852 THEN
				udiStatus2	:= 10028;	//Receive RevokeMachineReady While Downstream In Service Description State
			ELSIF udiStatus2 = 2853 THEN
				udiStatus2	:= 10029;	//Receive StartTransport While Downstream In Service Description State
			ELSIF udiStatus2 = 2854 THEN
				udiStatus2	:= 10030;	//Receive StopTransport While Downstream In Service Description State
			ELSIF udiStatus2 = 2855 THEN
				udiStatus2	:= 10031;	//Receive TransportFinished While Downstream In Service Description State
			ELSIF udiStatus2 = 2856 THEN
				udiStatus2	:= 10032;	//Receive BoardForecast While Downstream In Service Description State
			ELSIF udiStatus2 = 2857 THEN
				udiStatus2	:= 10033;	//Receive ServiceDescription While Downstream In Not Available Not Ready State
			ELSIF udiStatus2 = 2858 THEN
				udiStatus2	:= 10034;	//Receive BoardAvailable While Downstream In Not Available Not Ready State
			ELSIF udiStatus2 = 2859 THEN
				udiStatus2	:= 10035;	//Receive RevokeBoardAvailable While Downstream In Not Available Not Ready State
			ELSIF udiStatus2 = 2860 THEN
				udiStatus2	:= 10036;	//Receive RevokeMachineReady While Downstream In Not Available Not Ready State
			ELSIF udiStatus2 = 2861 THEN
				udiStatus2	:= 10037;	//Receive StartTransport While Downstream In Not Available Not Ready State
			ELSIF udiStatus2 = 2862 THEN
				udiStatus2	:= 10038;	//Receive StopTransport While Downstream In Not Available Not Ready State
			ELSIF udiStatus2 = 2863 THEN
				udiStatus2	:= 10039;	//Receive TransportFinished While Downstream In Not Available Not Ready State
			ELSIF udiStatus2 = 2864 THEN
				udiStatus2	:= 10040;	//Receive BoardForecast While Downstream In Not Available Not Ready State
			ELSIF udiStatus2 = 2865 THEN
				udiStatus2	:= 10041;	//Receive ServiceDescription While Downstream In Board Available State
			ELSIF udiStatus2 = 2866 THEN
				udiStatus2	:= 10042;	//Receive BoardAvailable While Downstream In Board Available State
			ELSIF udiStatus2 = 2867 THEN
				udiStatus2	:= 10043;	//Receive RevokeBoardAvailable While Downstream In Board Available State
			ELSIF udiStatus2 = 2868 THEN
				udiStatus2	:= 10044;	//Receive RevokeMachineReady While Downstream In Board Available State
			ELSIF udiStatus2 = 2869 THEN
				udiStatus2	:= 10045;	//Receive StartTransport While Downstream In Board Available State
			ELSIF udiStatus2 = 2870 THEN
				udiStatus2	:= 10046;	//Receive StopTransport While Downstream In Board Available State
			ELSIF udiStatus2 = 2871 THEN
				udiStatus2	:= 10047;	//Receive TransportFinished While Downstream In Board Available State
			ELSIF udiStatus2 = 2872 THEN
				udiStatus2	:= 10048;	//Receive BoardForecast While Downstream In Board Available State
			ELSIF udiStatus2 = 2873 THEN
				udiStatus2	:= 10049;	//Receive ServiceDescription While Downstream In Machine Ready State
			ELSIF udiStatus2 = 2874 THEN
				udiStatus2	:= 10050;	//Receive BoardAvailable While Downstream In Machine Ready State
			ELSIF udiStatus2 = 2875 THEN
				udiStatus2	:= 10051;	//Receive RevokeBoardAvailable While Downstream In Machine Ready State
			ELSIF udiStatus2 = 2876 THEN
				udiStatus2	:= 10052;	//Receive MachineReady While Downstream In Machine Ready State
			ELSIF udiStatus2 = 2877 THEN
				udiStatus2	:= 10053;	//Receive StopTransport While Downstream In Machine Ready State
			ELSIF udiStatus2 = 2878 THEN
				udiStatus2	:= 10054;	//Receive TransportFinished While Downstream In Machine Ready State
			ELSIF udiStatus2 = 2879 THEN
				udiStatus2	:= 10055;	//Receive BoardForecast While Downstream In Machine Ready State
			ELSIF udiStatus2 = 2880 THEN
				udiStatus2	:= 10056;	//Receive ServiceDescription While Downstream In Available And Ready State
			ELSIF udiStatus2 = 2881 THEN
				udiStatus2	:= 10057;	//Receive BoardAvailable While Downstream In Available And Ready State
			ELSIF udiStatus2 = 2882 THEN
				udiStatus2	:= 10058;	//Receive RevokeBoardAvailable While Downstream In Available And Ready State
			ELSIF udiStatus2 = 2883 THEN
				udiStatus2	:= 10059;	//Receive MachineReady While Downstream In Available And Ready State
			ELSIF udiStatus2 = 2884 THEN
				udiStatus2	:= 10060;	//Receive StopTransport While Downstream In Available And Ready State
			ELSIF udiStatus2 = 2885 THEN
				udiStatus2	:= 10061;	//Receive TransportFinished While Downstream In Available And Ready State
			ELSIF udiStatus2 = 2886 THEN
				udiStatus2	:= 10062;	//Receive BoardForecast While Downstream In Available And Ready State
			ELSIF udiStatus2 = 2887 THEN
				udiStatus2	:= 10063;	//Receive ServiceDescription While Downstream In Transporting State
			ELSIF udiStatus2 = 2888 THEN
				udiStatus2	:= 10064;	//Receive BoardAvailable While Downstream In Transporting State
			ELSIF udiStatus2 = 2889 THEN
				udiStatus2	:= 10065;	//Receive RevokeBoardAvailable While Downstream In Transporting State
			ELSIF udiStatus2 = 2890 THEN
				udiStatus2	:= 10066;	//Receive MachineReady While Downstream In Transporting State
			ELSIF udiStatus2 = 2891 THEN
				udiStatus2	:= 10067;	//Receive RevokeMachineReady While Downstream In Transporting State
			ELSIF udiStatus2 = 2892 THEN
				udiStatus2	:= 10068;	//Receive StartTransport While Downstream In Transporting State
			ELSIF udiStatus2 = 2893 THEN
				udiStatus2	:= 10069;	//Receive TransportFinished While Downstream In Transporting State
			ELSIF udiStatus2 = 2894 THEN
				udiStatus2	:= 10070;	//Receive BoardForecast While Downstream In Transporting State
			ELSIF udiStatus2 = 2895 THEN
				udiStatus2	:= 10071;	//Receive ServiceDescription While In Transport Finished State
			ELSIF udiStatus2 = 2896 THEN
				udiStatus2	:= 10072;	//Receive BoardAvailable While In Transport Finished State
			ELSIF udiStatus2 = 2897 THEN
				udiStatus2	:= 10073;	//Receive RevokeBoardAvailable While In Transport Finished State
			ELSIF udiStatus2 = 2898 THEN
				udiStatus2	:= 10074;	//Receive MachineReady While In Transport Finished State
			ELSIF udiStatus2 = 2899 THEN
				udiStatus2	:= 10075;	//Receive RevokeMachineReady While In Transport Finished State
			ELSIF udiStatus2 = 2900 THEN
				udiStatus2	:= 10076;	//Receive StartTransport While In Transport Finished State
			ELSIF udiStatus2 = 2901 THEN
				udiStatus2	:= 10077;	//Receive TransportFinished While In Transport Finished State
			ELSIF udiStatus2 = 2902 THEN
				udiStatus2	:= 10078;	//Receive BoardForecast While In Transport Finished State
			ELSIF udiStatus2 = 2903 THEN
				udiStatus2	:= 10079;	//Receive ServiceDescription While Downstream In Transport Stopped State
			ELSIF udiStatus2 = 2904 THEN
				udiStatus2	:= 10080;	//Receive BoardAvailable While Downstream In Transport Stopped State
			ELSIF udiStatus2 = 2905 THEN
				udiStatus2	:= 10081;	//Receive RevokeBoardAvailable While Downstream In Transport Stopped State
			ELSIF udiStatus2 = 2906 THEN
				udiStatus2	:= 10082;	//Receive MachineReady While Downstream In Transport Stopped State
			ELSIF udiStatus2 = 2907 THEN
				udiStatus2	:= 10083;	//Receive RevokeMachineReady While Downstream In Transport Stopped State
			ELSIF udiStatus2 = 2908 THEN
				udiStatus2	:= 10084;	//Receive StartTransport While Downstream In Transport Stopped State
			ELSIF udiStatus2 = 2909 THEN
				udiStatus2	:= 10085;	//Receive StopTransport While Downstream In Transport Stopped State
			ELSIF udiStatus2 = 2910 THEN
				udiStatus2	:= 10108;	//Receive TransportFinished While Downstream In Transport Stopped State
			ELSIF udiStatus2 = 2911 THEN
				udiStatus2	:= 10109;	//Receive BoardForecast While Downstream In Transport Stopped State
			END_IF

			fHermesAddOneMsgSend(ADR(a_eMsgSend) , ADR(udiMsgSendBffr) , HermesMsgTypeNotification);

			tyNotificationSnd.tyAvl.bSeverity			:= TRUE;
			tyNotificationSnd.tyAvl.bNotificationCode	:= TRUE;
			tyNotificationSnd.tyAvl.bDescription		:= TRUE;
			tyNotificationSnd.tyData.eSeverity			:= HermesSeverityFatalError;
			tyNotificationSnd.tyData.iNotificationCode	:= UDINT_TO_INT(udiStatus2);
			tyNotificationSnd.tyData.sDescription		:= a_tyAlmText[udiStatus2].sAlmText;

		END_IF

	END_IF

END_ACTION
```

#### Act_Background_NotificationRcv.st
```iecst
(** 2021-08-01 **)
ACTION Act_Background_NotificationRcv:

	IF eStatus1 <> Error THEN

		IF tyMsgTypeRcv.bNotification = TRUE THEN
			tyMsgTypeRcv.bNotification	:= FALSE;

			bRstConnection	:= fHermesNotificationRstConn(tyNotificationRcv) OR bRstConnection;
//			bRstState		:= fHermesNotificationRstState(tyNotificationRcv) OR bRstState;

		END_IF

	END_IF

END_ACTION
```

#### Act_Background_NotificationSnd.st
```iecst
(** 2019-03-15 **)
ACTION Act_Background_NotificationSnd:

	IF a_eMsgSend[0] = HermesMsgTypeNotification THEN
		bRstConnection	:= fHermesNotificationRstConn(tyNotificationSnd) OR bRstConnection;
//		bRstState		:= fHermesNotificationRstState(tyNotificationSnd) OR bRstState;
	END_IF

END_ACTION
```

#### Act_Background_Sequence.st
```iecst
 (** 2019-05-04 **)
ACTION Act_Background_Sequence:

	IF eStatus1 <> Error THEN

		IF p_bOpsRun = FALSE THEN
			p_bSndIncompl	:= TRUE;
		END_IF

		IF tyMsgTypeRcv.bStopTransport = TRUE THEN
			IF tyStopTransport.tyData.eTransferState = HermesTransferStateNotStarted THEN
				p_bSndNotStart	:= TRUE;
			ELSIF tyStopTransport.tyData.eTransferState = HermesTransferStateIncomplete THEN
				p_bSndIncompl	:= TRUE;
			END_IF
		END_IF

		bBlkDS := NOT(p_bHermesSwitchtoRvrseTransport);
		//Sequence
		fbSequenceDS.bRstState		:= bRstState;
		fbSequenceDS.bRdySnd		:= p_bRdySnd;
		fbSequenceDS.bBlkDS			:= bBlkDS;
		fbSequenceDS.bSndCompl		:= p_bSndCompl;
		fbSequenceDS.bSndIncompl	:= p_bSndIncompl;
		fbSequenceDS.bSndNotStart	:= p_bSndNotStart;
		fbSequenceDS.bFeatureBoardForecast	:= bFeatureBoardForecast; //Feature BoardForecast
		fbSequenceDS.bOpsRun	        	:= p_bOpsRun; //Machine in AutoMode
		fbSequenceDS.bSendBFId              := bSendBFId; //Send B.F with forecast ID, then block Hermes.eState until Downstream reply a MachineReady(Id) or MachineReady()
		fbSequenceDS.bBFIdSent              := bBFIdSent;
		fbSequenceDS.bSendBFNoID			:= bSendBFNoID;
		fbSequenceDS(bEn := TRUE);
		bUSRdy			:= fbSequenceDS.bUSRdy;
		bDSRdy			:= fbSequenceDS.bDSRdy;
		bTransporting	:= fbSequenceDS.bTransporting;
		bStopTransport	:= fbSequenceDS.bStopTransport;

		bUSGdRdy	:= (tyBoardAvailableSnd.tyAvl.bFailedBoard = FALSE) OR ((tyBoardAvailableSnd.tyAvl.bFailedBoard = TRUE) AND (tyBoardAvailableSnd.tyData.eFailedBoard <> HermesFailedBoard));

		bDSGdRdy	:= (tyMachineReady.tyAvl.bFailedBoard = FALSE) OR ((tyMachineReady.tyAvl.bFailedBoard = TRUE) AND (tyMachineReady.tyData.eFailedBoard <> HermesFailedBoard));

		IF fbSequenceDS.eState >= HermesStateNotAvailableNotReady THEN
			bHandshakeDone	:= TRUE;
		ELSE
			bHandshakeDone	:= FALSE;
		END_IF

		IF EDGEPOS(fbSequenceDS.eState = HermesStateTransporting) THEN
			p_bSndCompl		:= FALSE;
			p_bSndIncompl	:= FALSE;
			p_bSndNotStart	:= FALSE;
		END_IF

		IF fbSequenceDS.eMsgTypeSnd = HermesMsgTypeServiceDescription THEN
			fHermesAddOneMsgSend(ADR(a_eMsgSend) , ADR(udiMsgSendBffr) , HermesMsgTypeServiceDescription);

			tyServiceDescriptionSnd.tyData.sMachineId								    	:= p_sMcId;
			tyServiceDescriptionSnd.tyData.iLaneId											:= p_tyParam.iLaneID;
			tyServiceDescriptionSnd.tyData.sInterfaceId										:= p_sInterfaceId;
			tyServiceDescriptionSnd.tyData.sVersion											:= p_sVersion;
			tyServiceDescriptionSnd.tyData.tySupportedFeatures.bFeatureCheckAliveResponse	:= (p_tyParam.bFeatureCheckAliveResponse) AND (p_tyParam.tRcvAlive <> T#0s) AND (p_tyParam.tSndAlive <> T#0s);
			tyServiceDescriptionSnd.tyData.tySupportedFeatures.bFeatureBoardForecast		:= p_tyParam.bFeatureBoardForecast;
			tyServiceDescriptionSnd.tyData.tySupportedFeatures.bFeatureQueryBoardInfo		:= FALSE;
			tyServiceDescriptionSnd.tyData.tySupportedFeatures.bFeatureSendBoardInfo		:= p_tyParam.bFeatureSendBoardInfo;
			tyServiceDescriptionSnd.tyData.tySupportedFeatures.bFeatureCommand				:= p_tyParam.bFeatureCommand;

			tyServiceDescriptionSnd.tyAvl.bMachineId										:= tyServiceDescriptionSnd.tyData.sMachineId <> '';
			tyServiceDescriptionSnd.tyAvl.bLaneId											:= tyServiceDescriptionSnd.tyData.iLaneId<>0;
			tyServiceDescriptionSnd.tyAvl.bInterfaceId										:= tyServiceDescriptionSnd.tyData.sInterfaceId <> '';
			tyServiceDescriptionSnd.tyAvl.bVersion											:= TRUE;
			tyServiceDescriptionSnd.tyAvl.bSupportedFeatures								:= p_tyParam.bFeatureCheckAliveResponse OR p_tyParam.bFeatureBoardForecast OR p_tyParam.bFeatureSendBoardInfo OR p_tyParam.bFeatureCommand;
			tyServiceDescriptionSnd.tyAvl.tySupportedFeatures.bFeatureCheckAliveResponse	:= (p_tyParam.bFeatureCheckAliveResponse) AND (p_tyParam.tRcvAlive <> T#0s) AND (p_tyParam.tSndAlive <> T#0s);
			tyServiceDescriptionSnd.tyAvl.tySupportedFeatures.bFeatureBoardForecast			:= p_tyParam.bFeatureBoardForecast;
			tyServiceDescriptionSnd.tyAvl.tySupportedFeatures.bFeatureQueryBoardInfo		:= FALSE;
			tyServiceDescriptionSnd.tyAvl.tySupportedFeatures.bFeatureSendBoardInfo			:= p_tyParam.bFeatureSendBoardInfo;
			tyServiceDescriptionSnd.tyAvl.tySupportedFeatures.bFeatureCommand				:= p_tyParam.bFeatureCommand;
		ELSIF fbSequenceDS.eMsgTypeSnd = HermesMsgTypeBoardForecastId THEN //Properties changed
			//need to mantain at one
			fHermesAddOneMsgSend(ADR(a_eMsgSend) , ADR(udiMsgSendBffr) , HermesMsgTypeBoardForecast);
			fHermesGenerateUUID(ADR(tyBoardForecastSnd.tyData.sForecastId) , p_tyDTStructure , pa_usiMacAddr); //Generate ForecastID if there is new Product Changeover
			bBFIdSent := TRUE;

			IF p_bManualInsertData = FALSE THEN //insert board function (from SvyHermes)
				tyBoardForecastSnd.tyData.rTimeUntilAvailable       := p_rMcCycleTm + p_rAWCycleTm;
				tyBoardForecastSnd.tyData.sBoardId 			        := ''; //no need to send BoardId for HermesMsgTypeBoardForecastId.
				tyBoardForecastSnd.tyData.sBoardIdCreatedBy			:= ''; //no need to send BoardIdCreatedBy since no BoardId.
				tyBoardForecastSnd.tyData.eFailedBoard 			    := p_eFailedBoard;
				tyBoardForecastSnd.tyData.sProductTypeId 			:= p_sRecipeNm; //recipe0 name = running recipe name
				tyBoardForecastSnd.tyData.eFlippedBoard 			:= p_eFlippedBoard;
				tyBoardForecastSnd.tyData.sTopBarcode 		    	:= p_sTopBarcode;
				tyBoardForecastSnd.tyData.sBottomBarcode 			:= p_sBottomBarcode;
				tyBoardForecastSnd.tyData.rLength 				    := p_rLength;
				tyBoardForecastSnd.tyData.rWidth 			    	:= DINT_TO_REAL(p_diWidthInUM) / 1000; //recipe 0 width	 = running recipe width
				tyBoardForecastSnd.tyData.rThickness 		    	:= p_rThickness;
				tyBoardForecastSnd.tyData.rConveyorSpeed 			:= p_rConveyorSpeed;
				tyBoardForecastSnd.tyData.rTopClearanceHeight 		:= p_rTopClearanceHeight;
				tyBoardForecastSnd.tyData.rBottomClearanceHeight 	:= p_rBottomClearanceHeight;
				tyBoardForecastSnd.tyData.rWeight 			    	:= p_rWeight;
				tyBoardForecastSnd.tyData.sWorkOrderId 			    := p_sWorkOrderId;
				tyBoardForecastSnd.tyData.sBatchId 			        := p_sBatchId;

				tyBoardForecastSnd.tyAvl.bForecastId 			    := TRUE;
				tyBoardForecastSnd.tyAvl.bTimeUntilAvailable		:= tyBoardForecastSnd.tyData.rTimeUntilAvailable <> 0;
				tyBoardForecastSnd.tyAvl.bBoardId 				    := tyBoardForecastSnd.tyData.sBoardId <> '';
				tyBoardForecastSnd.tyAvl.bBoardIdCreatedBy 		    := TRUE;
				tyBoardForecastSnd.tyAvl.bFailedBoard 			    := TRUE;
				tyBoardForecastSnd.tyAvl.bProductTypeId 			:= tyBoardForecastSnd.tyData.sProductTypeId <> '';
				tyBoardForecastSnd.tyAvl.bFlippedBoard 			    := TRUE;
				tyBoardForecastSnd.tyAvl.bTopBarcode 			    := tyBoardForecastSnd.tyData.sTopBarcode <> '';
				tyBoardForecastSnd.tyAvl.bBottomBarcode 			:= tyBoardForecastSnd.tyData.sBottomBarcode <> '';
				tyBoardForecastSnd.tyAvl.bLength 				    := tyBoardForecastSnd.tyData.rLength <> 0;
				tyBoardForecastSnd.tyAvl.bWidth 				    := tyBoardForecastSnd.tyData.rWidth <> 0 AND (p_bBFWidthEn = TRUE);
				tyBoardForecastSnd.tyAvl.bThickness 			    := tyBoardForecastSnd.tyData.rThickness <> 0 AND (p_bBFSltEn = TRUE);
				tyBoardForecastSnd.tyAvl.bConveyorSpeed 			:= tyBoardForecastSnd.tyData.rConveyorSpeed <> 0;
				tyBoardForecastSnd.tyAvl.bTopClearanceHeight 		:= tyBoardForecastSnd.tyData.rTopClearanceHeight <> 0 AND (p_bBFSltEn = TRUE);
				tyBoardForecastSnd.tyAvl.bBottomClearanceHeight 	:= tyBoardForecastSnd.tyData.rBottomClearanceHeight <> 0 AND (p_bBFSltEn = TRUE);
				tyBoardForecastSnd.tyAvl.bWeight 			    	:= tyBoardForecastSnd.tyData.rWeight <> 0;
				tyBoardForecastSnd.tyAvl.bWorkOrderId 		    	:= tyBoardForecastSnd.tyData.sWorkOrderId <> '';
				tyBoardForecastSnd.tyAvl.bBatchId 		        	:= tyBoardForecastSnd.tyData.sBatchId <> '';
			ELSE //from Rcp
				tyBoardForecastSnd.tyData.rTimeUntilAvailable       := p_rMcCycleTm + p_rAWCycleTm;
				tyBoardForecastSnd.tyData.sBoardId 			        := ''; //no need to send BoardId for HermesMsgTypeBoardForecastId.
				tyBoardForecastSnd.tyData.sBoardIdCreatedBy			:= ''; //no need to send BoardIdCreatedBy since no BoardId.
				tyBoardForecastSnd.tyData.eFailedBoard 			    := p_tySvyHermesSendWorkOrderInfo.tyData.eFailedBoard;
				tyBoardForecastSnd.tyData.sProductTypeId 			:= p_tySvyHermesSendWorkOrderInfo.tyData.sProductTypeId;
				tyBoardForecastSnd.tyData.eFlippedBoard 			:= p_tySvyHermesSendWorkOrderInfo.tyData.eFlippedBoard;
				tyBoardForecastSnd.tyData.sTopBarcode 		    	:= p_tySvyHermesSendWorkOrderInfo.tyData.sTopBarcode;
				tyBoardForecastSnd.tyData.sBottomBarcode 			:= p_tySvyHermesSendWorkOrderInfo.tyData.sBottomBarcode;
				tyBoardForecastSnd.tyData.rLength 				    := p_tySvyHermesSendWorkOrderInfo.tyData.rLength;
				tyBoardForecastSnd.tyData.rWidth 			    	:= DINT_TO_REAL(p_diWidthInUM) / 1000; //recipe 0 width	 = running recipe width
				tyBoardForecastSnd.tyData.rThickness 		    	:= p_tySvyHermesSendWorkOrderInfo.tyData.rThickness;
				tyBoardForecastSnd.tyData.rConveyorSpeed 			:= p_tySvyHermesSendWorkOrderInfo.tyData.rConveyorSpeed;
				tyBoardForecastSnd.tyData.rTopClearanceHeight 		:= p_tySvyHermesSendWorkOrderInfo.tyData.rTopClearanceHeight;
				tyBoardForecastSnd.tyData.rBottomClearanceHeight 	:= p_tySvyHermesSendWorkOrderInfo.tyData.rBottomClearanceHeight;
				tyBoardForecastSnd.tyData.rWeight 			    	:= p_tySvyHermesSendWorkOrderInfo.tyData.rWeight;
				tyBoardForecastSnd.tyData.sWorkOrderId 			    := p_tySvyHermesSendWorkOrderInfo.tyData.sWorkOrderId;
				tyBoardForecastSnd.tyData.sBatchId 			        := p_tySvyHermesSendWorkOrderInfo.tyData.sBatchId;

				tyBoardForecastSnd.tyAvl.bForecastId 			    := TRUE;
				tyBoardForecastSnd.tyAvl.bTimeUntilAvailable		:= tyBoardForecastSnd.tyData.rTimeUntilAvailable <> 0;
				tyBoardForecastSnd.tyAvl.bBoardId 				    := tyBoardForecastSnd.tyData.sBoardId <> '';
				tyBoardForecastSnd.tyAvl.bBoardIdCreatedBy 		    := TRUE;
				tyBoardForecastSnd.tyAvl.bFailedBoard 			    := TRUE;
				tyBoardForecastSnd.tyAvl.bProductTypeId 			:= tyBoardForecastSnd.tyData.sProductTypeId <> '';
				tyBoardForecastSnd.tyAvl.bFlippedBoard 			    := TRUE;
				tyBoardForecastSnd.tyAvl.bTopBarcode 			    := tyBoardForecastSnd.tyData.sTopBarcode <> '';
				tyBoardForecastSnd.tyAvl.bBottomBarcode 			:= tyBoardForecastSnd.tyData.sBottomBarcode <> '';
				tyBoardForecastSnd.tyAvl.bLength 				    := tyBoardForecastSnd.tyData.rLength <> 0;
				tyBoardForecastSnd.tyAvl.bWidth 				    := tyBoardForecastSnd.tyData.rWidth <> 0 AND (p_bBFWidthEn = TRUE);
				tyBoardForecastSnd.tyAvl.bThickness 			    := tyBoardForecastSnd.tyData.rThickness <> 0 AND (p_bBFSltEn = TRUE);
				tyBoardForecastSnd.tyAvl.bConveyorSpeed 			:= tyBoardForecastSnd.tyData.rConveyorSpeed <> 0;
				tyBoardForecastSnd.tyAvl.bTopClearanceHeight 		:= tyBoardForecastSnd.tyData.rTopClearanceHeight <> 0 AND (p_bBFSltEn = TRUE);
				tyBoardForecastSnd.tyAvl.bBottomClearanceHeight 	:= tyBoardForecastSnd.tyData.rBottomClearanceHeight <> 0 AND (p_bBFSltEn = TRUE);
				tyBoardForecastSnd.tyAvl.bWeight 			    	:= tyBoardForecastSnd.tyData.rWeight <> 0;
				tyBoardForecastSnd.tyAvl.bWorkOrderId 		    	:= tyBoardForecastSnd.tyData.sWorkOrderId <> '';
				tyBoardForecastSnd.tyAvl.bBatchId 		        	:= tyBoardForecastSnd.tyData.sBatchId <> '';

			END_IF

		ELSIF fbSequenceDS.eMsgTypeSnd = HermesMsgTypeBoardForecastNoId THEN
			//do not need to count
			fHermesAddOneMsgSend(ADR(a_eMsgSend) , ADR(udiMsgSendBffr) , HermesMsgTypeBoardForecast);
			tyBoardForecastSnd.tyData.sForecastId		        := ''; //Do not need to generate ForecastID to downstream

			IF p_bNewBrdAvlFirstZone AND p_usiUSHermesReverseDSSendBFId <> 0 THEN //Tigger by US hermes to Reverse DS Hermes

				IF p_usiUSHermesReverseDSSendBFId = 1 THEN //up pulse trigger with BrdId
					fbParseBrdAvlExternal.p_XMLTable		:= ADR(pa_RevtyXMLTableDataBrdAvl);//last zone B.A
					fbParseBrdAvlExternal.iTotalIdxWrite	:= p_ReviXMLTableDataBrdAvlTtlIdx; //last zone
					fbParseBrdAvlExternal;
					fHermesBrdAvltoBF(ADR(tyBoardForecastSnd),ADR(fbParseBrdAvlExternal.tyBoardAvailable));
				ELSIF p_usiUSHermesReverseDSSendBFId = 2 THEN  //downpulse , reset
					memset(ADR(tyBoardForecastSnd),0,SIZEOF(tyBoardForecastSnd));

					tyBoardForecastSnd.tyAvl.bFailedBoard 			    := TRUE;
					tyBoardForecastSnd.tyAvl.bFlippedBoard 			    := TRUE;
				END_IF
			ELSIF p_bNewBrdAvlFirstZone AND p_bManualInsertData = FALSE THEN
				fHermesGenerateUUID(ADR(tyBoardForecastSnd.tyData.sBoardId) , p_tyDTStructure , pa_usiMacAddr);
				tyBoardForecastSnd.tyData.sBoardIdCreatedBy         := p_sMcId;
				tyBoardForecastSnd.tyData.eFailedBoard 		    	:= p_eFailedBoard;
				tyBoardForecastSnd.tyData.sProductTypeId 			:= p_sRecipeNm;	 //recipe 0 name = running recipe name
				tyBoardForecastSnd.tyData.eFlippedBoard 			:= p_eFlippedBoard;
				tyBoardForecastSnd.tyData.sTopBarcode 		    	:= p_sTopBarcode;
				tyBoardForecastSnd.tyData.sBottomBarcode 			:= p_sBottomBarcode;
				tyBoardForecastSnd.tyData.rLength 				    := p_rLength;
				tyBoardForecastSnd.tyData.rWidth 			    	:= DINT_TO_REAL(p_diWidthInUM) / 1000;	//recipe 0 width = running recipe width
				tyBoardForecastSnd.tyData.rThickness 		    	:= p_rThickness;
				tyBoardForecastSnd.tyData.rConveyorSpeed 			:= p_rConveyorSpeed;
				tyBoardForecastSnd.tyData.rTopClearanceHeight 		:= p_rTopClearanceHeight;
				tyBoardForecastSnd.tyData.rBottomClearanceHeight 	:= p_rBottomClearanceHeight;
				tyBoardForecastSnd.tyData.rWeight 			    	:= p_rWeight;
				tyBoardForecastSnd.tyData.sWorkOrderId 		    	:= p_sWorkOrderId;
				tyBoardForecastSnd.tyData.sBatchId	    	    	:= p_sBatchId;

				tyBoardForecastSnd.tyAvl.bForecastId 			    := tyBoardForecastSnd.tyData.sForecastId <> '';
				tyBoardForecastSnd.tyAvl.bTimeUntilAvailable		:= tyBoardForecastSnd.tyData.rTimeUntilAvailable <> 0;
				tyBoardForecastSnd.tyAvl.bBoardId 				    := tyBoardForecastSnd.tyData.sBoardId <> '';
				tyBoardForecastSnd.tyAvl.bBoardIdCreatedBy 	    	:= tyBoardForecastSnd.tyData.sBoardIdCreatedBy <> '';
				tyBoardForecastSnd.tyAvl.bFailedBoard 			    := TRUE;
				tyBoardForecastSnd.tyAvl.bProductTypeId 			:= tyBoardForecastSnd.tyData.sProductTypeId <> '';
				tyBoardForecastSnd.tyAvl.bFlippedBoard 		    	:= TRUE;
				tyBoardForecastSnd.tyAvl.bTopBarcode 			    := tyBoardForecastSnd.tyData.sTopBarcode <> '';
				tyBoardForecastSnd.tyAvl.bBottomBarcode 			:= tyBoardForecastSnd.tyData.sBottomBarcode <> '';
				tyBoardForecastSnd.tyAvl.bLength 				    := tyBoardForecastSnd.tyData.rLength <> 0;
				tyBoardForecastSnd.tyAvl.bWidth 				    := tyBoardForecastSnd.tyData.rWidth <> 0 AND (p_bBFWidthEn = TRUE);
				tyBoardForecastSnd.tyAvl.bThickness 			    := tyBoardForecastSnd.tyData.rThickness <> 0 AND (p_bBFSltEn = TRUE);
				tyBoardForecastSnd.tyAvl.bConveyorSpeed 			:= tyBoardForecastSnd.tyData.rConveyorSpeed <> 0;
				tyBoardForecastSnd.tyAvl.bTopClearanceHeight 		:= tyBoardForecastSnd.tyData.rTopClearanceHeight <>0 AND (p_bBFSltEn = TRUE);
				tyBoardForecastSnd.tyAvl.bBottomClearanceHeight 	:= tyBoardForecastSnd.tyData.rBottomClearanceHeight <>0 AND (p_bBFSltEn = TRUE);
				tyBoardForecastSnd.tyAvl.bWeight 			    	:= tyBoardForecastSnd.tyData.rWeight <> 0;
				tyBoardForecastSnd.tyAvl.bWorkOrderId 		    	:= tyBoardForecastSnd.tyData.sWorkOrderId <> '';
				tyBoardForecastSnd.tyAvl.bBatchId 		        	:= tyBoardForecastSnd.tyData.sBatchId <> '';
			ELSIF p_bNewBrdAvlFirstZone AND p_bManualInsertData THEN //insert board data
				fHermesGenerateUUID(ADR(tyBoardForecastSnd.tyData.sBoardId) , p_tyDTStructure , pa_usiMacAddr);
				tyBoardForecastSnd.tyData.sBoardIdCreatedBy         := p_sMcId;
				tyBoardForecastSnd.tyData.eFailedBoard 		    	:= p_tySvyHermesSendWorkOrderInfo.tyData.eFailedBoard;
				tyBoardForecastSnd.tyData.sProductTypeId 			:= p_tySvyHermesSendWorkOrderInfo.tyData.sProductTypeId;
				tyBoardForecastSnd.tyData.eFlippedBoard 			:= p_tySvyHermesSendWorkOrderInfo.tyData.eFlippedBoard;
				tyBoardForecastSnd.tyData.sTopBarcode 		    	:= p_tySvyHermesSendWorkOrderInfo.tyData.sTopBarcode;
				tyBoardForecastSnd.tyData.sBottomBarcode 			:= p_tySvyHermesSendWorkOrderInfo.tyData.sBottomBarcode;
				tyBoardForecastSnd.tyData.rLength 				    := p_tySvyHermesSendWorkOrderInfo.tyData.rLength;
				tyBoardForecastSnd.tyData.rWidth 			    	:= DINT_TO_REAL(p_diWidthInUM) / 1000;	//recipe 0 width = running recipe width
				tyBoardForecastSnd.tyData.rThickness 		    	:= p_tySvyHermesSendWorkOrderInfo.tyData.rThickness;
				tyBoardForecastSnd.tyData.rConveyorSpeed 			:= p_tySvyHermesSendWorkOrderInfo.tyData.rConveyorSpeed;
				tyBoardForecastSnd.tyData.rTopClearanceHeight 		:= p_tySvyHermesSendWorkOrderInfo.tyData.rTopClearanceHeight;
				tyBoardForecastSnd.tyData.rBottomClearanceHeight 	:= p_tySvyHermesSendWorkOrderInfo.tyData.rBottomClearanceHeight;
				tyBoardForecastSnd.tyData.rWeight 			    	:= p_tySvyHermesSendWorkOrderInfo.tyData.rWeight;
				tyBoardForecastSnd.tyData.sWorkOrderId 		    	:= p_tySvyHermesSendWorkOrderInfo.tyData.sWorkOrderId;
				tyBoardForecastSnd.tyData.sBatchId	    	    	:= p_tySvyHermesSendWorkOrderInfo.tyData.sBatchId;

				tyBoardForecastSnd.tyAvl.bForecastId 			    := tyBoardForecastSnd.tyData.sForecastId <> '';
				tyBoardForecastSnd.tyAvl.bTimeUntilAvailable		:= tyBoardForecastSnd.tyData.rTimeUntilAvailable <> 0;
				tyBoardForecastSnd.tyAvl.bBoardId 				    := tyBoardForecastSnd.tyData.sBoardId <> '';
				tyBoardForecastSnd.tyAvl.bBoardIdCreatedBy 	    	:= tyBoardForecastSnd.tyData.sBoardIdCreatedBy <> '';
				tyBoardForecastSnd.tyAvl.bFailedBoard 			    := TRUE;
				tyBoardForecastSnd.tyAvl.bProductTypeId 			:= tyBoardForecastSnd.tyData.sProductTypeId <> '';
				tyBoardForecastSnd.tyAvl.bFlippedBoard 		    	:= TRUE;
				tyBoardForecastSnd.tyAvl.bTopBarcode 			    := tyBoardForecastSnd.tyData.sTopBarcode <> '';
				tyBoardForecastSnd.tyAvl.bBottomBarcode 			:= tyBoardForecastSnd.tyData.sBottomBarcode <> '';
				tyBoardForecastSnd.tyAvl.bLength 				    := tyBoardForecastSnd.tyData.rLength <> 0;
				tyBoardForecastSnd.tyAvl.bWidth 				    := tyBoardForecastSnd.tyData.rWidth <> 0 AND (p_bBFWidthEn = TRUE);
				tyBoardForecastSnd.tyAvl.bThickness 			    := tyBoardForecastSnd.tyData.rThickness <> 0 AND (p_bBFSltEn = TRUE);
				tyBoardForecastSnd.tyAvl.bConveyorSpeed 			:= tyBoardForecastSnd.tyData.rConveyorSpeed <> 0;
				tyBoardForecastSnd.tyAvl.bTopClearanceHeight 		:= tyBoardForecastSnd.tyData.rTopClearanceHeight <>0 AND (p_bBFSltEn = TRUE);
				tyBoardForecastSnd.tyAvl.bBottomClearanceHeight 	:= tyBoardForecastSnd.tyData.rBottomClearanceHeight <>0 AND (p_bBFSltEn = TRUE);
				tyBoardForecastSnd.tyAvl.bWeight 			    	:= tyBoardForecastSnd.tyData.rWeight <> 0;
				tyBoardForecastSnd.tyAvl.bWorkOrderId 		    	:= tyBoardForecastSnd.tyData.sWorkOrderId <> '';
				tyBoardForecastSnd.tyAvl.bBatchId 		        	:= tyBoardForecastSnd.tyData.sBatchId <> '';

			ELSE   //have brd detail

				//fBrdAvltoBFcast(ADR(),ADR());
				tyBoardForecastSnd.tyData.sBoardId                  := p_tyUSBoardArrivedData.tyData.sBoardId;
				tyBoardForecastSnd.tyData.sBoardIdCreatedBy         := p_tyUSBoardArrivedData.tyData.sBoardIdCreatedBy;
				tyBoardForecastSnd.tyData.eFailedBoard 		    	:= p_tyUSBoardArrivedData.tyData.eFailedBoard;
				tyBoardForecastSnd.tyData.sProductTypeId 			:= p_tyUSBoardArrivedData.tyData.sProductTypeId;
				tyBoardForecastSnd.tyData.eFlippedBoard 			:= p_tyUSBoardArrivedData.tyData.eFlippedBoard;
				tyBoardForecastSnd.tyData.sTopBarcode 		    	:= p_tyUSBoardArrivedData.tyData.sTopBarcode;
				tyBoardForecastSnd.tyData.sBottomBarcode 			:= p_tyUSBoardArrivedData.tyData.sBottomBarcode;
				tyBoardForecastSnd.tyData.rLength 				    := p_tyUSBoardArrivedData.tyData.rLength;
				tyBoardForecastSnd.tyData.rWidth 			    	:= p_tyUSBoardArrivedData.tyData.rWidth;
				tyBoardForecastSnd.tyData.rThickness 		    	:= p_tyUSBoardArrivedData.tyData.rThickness;
				tyBoardForecastSnd.tyData.rConveyorSpeed 			:= p_tyUSBoardArrivedData.tyData.rConveyorSpeed;
				tyBoardForecastSnd.tyData.rTopClearanceHeight 		:= p_tyUSBoardArrivedData.tyData.rTopClearanceHeight;
				tyBoardForecastSnd.tyData.rBottomClearanceHeight 	:= p_tyUSBoardArrivedData.tyData.rBottomClearanceHeight;
				tyBoardForecastSnd.tyData.rWeight 			    	:= p_tyUSBoardArrivedData.tyData.rWeight;
				tyBoardForecastSnd.tyData.sWorkOrderId 		    	:= p_tyUSBoardArrivedData.tyData.sWorkOrderId;
				tyBoardForecastSnd.tyData.sBatchId 		        	:= p_tyUSBoardArrivedData.tyData.sBatchId;

				tyBoardForecastSnd.tyAvl.bForecastId 			    := tyBoardForecastSnd.tyData.sForecastId <> '';
				tyBoardForecastSnd.tyAvl.bTimeUntilAvailable		:= tyBoardForecastSnd.tyData.rTimeUntilAvailable <> 0;
				tyBoardForecastSnd.tyAvl.bBoardId 				    := tyBoardForecastSnd.tyData.sBoardId <> '';
				tyBoardForecastSnd.tyAvl.bBoardIdCreatedBy 	    	:= tyBoardForecastSnd.tyData.sBoardIdCreatedBy <> '';
				tyBoardForecastSnd.tyAvl.bFailedBoard 			    := TRUE;
				tyBoardForecastSnd.tyAvl.bProductTypeId 			:= tyBoardForecastSnd.tyData.sProductTypeId <> '';
				tyBoardForecastSnd.tyAvl.bFlippedBoard 		    	:= TRUE;
				tyBoardForecastSnd.tyAvl.bTopBarcode 			    := tyBoardForecastSnd.tyData.sTopBarcode <> '';
				tyBoardForecastSnd.tyAvl.bBottomBarcode 			:= tyBoardForecastSnd.tyData.sBottomBarcode <> '';
				tyBoardForecastSnd.tyAvl.bLength 				    := tyBoardForecastSnd.tyData.rLength <> 0;
				tyBoardForecastSnd.tyAvl.bWidth 				    := tyBoardForecastSnd.tyData.rWidth <> 0;
				tyBoardForecastSnd.tyAvl.bThickness 			    := tyBoardForecastSnd.tyData.rThickness <> 0;
				tyBoardForecastSnd.tyAvl.bConveyorSpeed 			:= tyBoardForecastSnd.tyData.rConveyorSpeed <> 0;
				tyBoardForecastSnd.tyAvl.bTopClearanceHeight 		:= tyBoardForecastSnd.tyData.rTopClearanceHeight <> 0;
				tyBoardForecastSnd.tyAvl.bBottomClearanceHeight 	:= tyBoardForecastSnd.tyData.rBottomClearanceHeight <> 0;
				tyBoardForecastSnd.tyAvl.bWeight 			    	:= tyBoardForecastSnd.tyData.rWeight <> 0;
				tyBoardForecastSnd.tyAvl.bWorkOrderId 		    	:= tyBoardForecastSnd.tyData.sWorkOrderId <> '';
				tyBoardForecastSnd.tyAvl.bBatchId 		        	:= tyBoardForecastSnd.tyData.sBatchId <> '';

			END_IF
		ELSIF fbSequenceDS.eMsgTypeSnd = HermesMsgTypeBoardAvailable THEN
			fHermesAddOneMsgSend(ADR(a_eMsgSend) , ADR(udiMsgSendBffr) , HermesMsgTypeBoardAvailable);

			tyBoardAvailableSnd.tyData.iRoute	:= iRoute;
			tyBoardAvailableSnd.tyData.iAction	:= iAction;

			tyBoardAvailableSnd.tyAvl.bRoute := tyBoardAvailableSnd.tyData.iRoute <> 0;
			tyBoardAvailableSnd.tyAvl.bAction:= tyBoardAvailableSnd.tyData.iAction <> 0 ;

			IF p_bNewBrdAvlLastZone = TRUE AND p_bRcvBoardInfo = FALSE THEN //Generate New B.A for Unknown PCB
				IF bFeatureBoardForecast AND bBFIdSent THEN
					tyBoardAvailableSnd.tyData.sBoardId :=	 tyBoardForecastSnd.tyData.sBoardId;
				ELSE
					fHermesGenerateUUID(ADR(tyBoardAvailableSnd.tyData.sBoardId) , p_tyDTStructure , pa_usiMacAddr);
				END_IF

				tyBoardAvailableSnd.tyData.sBoardIdCreatedBy        := p_sMcId; //Generate by our Machine
				tyBoardAvailableSnd.tyData.eFailedBoard				:= p_eFailedBoard;
				tyBoardAvailableSnd.tyData.sProductTypeId			:= p_sRecipeNm;
				tyBoardAvailableSnd.tyData.eFlippedBoard			:= p_eFlippedBoard;
				tyBoardAvailableSnd.tyData.sTopBarcode				:= p_sTopBarcode;
				tyBoardAvailableSnd.tyData.sBottomBarcode			:= p_sBottomBarcode;
				tyBoardAvailableSnd.tyData.rLength					:= p_rLength;
				tyBoardAvailableSnd.tyData.rWidth					:= DINT_TO_REAL(p_diWidthInUM) / 1000;
				tyBoardAvailableSnd.tyData.rThickness				:= p_rThickness;
				tyBoardAvailableSnd.tyData.rConveyorSpeed			:= p_rConveyorSpeed;
				tyBoardAvailableSnd.tyData.rTopClearanceHeight		:= p_rTopClearanceHeight;
				tyBoardAvailableSnd.tyData.rBottomClearanceHeight	:= p_rBottomClearanceHeight;
				tyBoardAvailableSnd.tyData.rWeight					:= p_rWeight;
				tyBoardAvailableSnd.tyData.sWorkOrderId			    := p_sWorkOrderId;
				tyBoardAvailableSnd.tyData.sBatchId			        := p_sBatchId;

				tyBoardAvailableSnd.tyAvl.bBoardId					:= tyBoardAvailableSnd.tyData.sBoardId<>'';
				tyBoardAvailableSnd.tyAvl.bBoardIdCreatedBy			:= tyBoardAvailableSnd.tyData.sBoardIdCreatedBy <> '';
				tyBoardAvailableSnd.tyAvl.bFailedBoard				:= TRUE;
				tyBoardAvailableSnd.tyAvl.bProductTypeId			:= tyBoardAvailableSnd.tyData.sProductTypeId <> '';
				tyBoardAvailableSnd.tyAvl.bFlippedBoard				:= TRUE;
				tyBoardAvailableSnd.tyAvl.bTopBarcode				:= tyBoardAvailableSnd.tyData.sTopBarcode <> '';
				tyBoardAvailableSnd.tyAvl.bBottomBarcode			:= tyBoardAvailableSnd.tyData.sBottomBarcode <> '';
				tyBoardAvailableSnd.tyAvl.bLength					:= tyBoardAvailableSnd.tyData.rLength <> 0;
				tyBoardAvailableSnd.tyAvl.bWidth					:= (tyBoardAvailableSnd.tyData.rWidth <> 0) AND (p_bBAWidthEn = TRUE);
				tyBoardAvailableSnd.tyAvl.bThickness				:= (tyBoardAvailableSnd.tyData.rThickness <> 0) AND (p_bBASltEn = TRUE);
				tyBoardAvailableSnd.tyAvl.bConveyorSpeed			:= tyBoardAvailableSnd.tyData.rConveyorSpeed <> 0;
				tyBoardAvailableSnd.tyAvl.bTopClearanceHeight		:= (tyBoardAvailableSnd.tyData.rTopClearanceHeight <> 0) AND (p_bBASltEn = TRUE);
				tyBoardAvailableSnd.tyAvl.bBottomClearanceHeight	:= (tyBoardAvailableSnd.tyData.rBottomClearanceHeight <> 0) AND (p_bBASltEn = TRUE);
				tyBoardAvailableSnd.tyAvl.bWeight					:= tyBoardAvailableSnd.tyData.rWeight <> 0;
				tyBoardAvailableSnd.tyAvl.bWorkOrderId				:= tyBoardAvailableSnd.tyData.sWorkOrderId <> '';
				tyBoardAvailableSnd.tyAvl.bBatchId			    	:= tyBoardAvailableSnd.tyData.sBatchId <> '';

			ELSIF p_bNewBrdAvlLastZone = TRUE AND p_bRcvBoardInfo = TRUE THEN //Take BoardInfo From "SendBoardInfo", for Manual Insert PCB

				tyBoardAvailableSnd.tyData.sBoardId                 := p_tyBoardInfoData.tyData.sBoardId;
				tyBoardAvailableSnd.tyData.sBoardIdCreatedBy        := p_tyBoardInfoData.tyData.sBoardIdCreatedBy;
				tyBoardAvailableSnd.tyData.eFailedBoard				:= p_tyBoardInfoData.tyData.eFailedBoard;
				tyBoardAvailableSnd.tyData.sProductTypeId			:= p_tyBoardInfoData.tyData.sProductTypeId;
				tyBoardAvailableSnd.tyData.eFlippedBoard			:= p_tyBoardInfoData.tyData.eFlippedBoard;
				tyBoardAvailableSnd.tyData.sTopBarcode				:= p_tyBoardInfoData.tyData.sTopBarcode;
				tyBoardAvailableSnd.tyData.sBottomBarcode			:= p_tyBoardInfoData.tyData.sBottomBarcode;
				tyBoardAvailableSnd.tyData.rLength					:= p_tyBoardInfoData.tyData.rLength;
				tyBoardAvailableSnd.tyData.rWidth					:= p_tyBoardInfoData.tyData.rWidth;
				tyBoardAvailableSnd.tyData.rThickness				:= p_tyBoardInfoData.tyData.rThickness;
				tyBoardAvailableSnd.tyData.rConveyorSpeed			:= p_rConveyorSpeed; //dont have
				tyBoardAvailableSnd.tyData.rTopClearanceHeight		:= p_tyBoardInfoData.tyData.rTopClearanceHeight;
				tyBoardAvailableSnd.tyData.rBottomClearanceHeight	:= p_tyBoardInfoData.tyData.rBottomClearanceHeight;
				tyBoardAvailableSnd.tyData.rWeight					:= p_tyBoardInfoData.tyData.rWeight;
				tyBoardAvailableSnd.tyData.sWorkOrderId			    := p_tyBoardInfoData.tyData.sWorkOrderId;
				tyBoardAvailableSnd.tyData.sBatchId		            := p_tyBoardInfoData.tyData.sBatchId;

				tyBoardAvailableSnd.tyAvl.bBoardId					:= tyBoardAvailableSnd.tyData.sBoardId <> '';
				tyBoardAvailableSnd.tyAvl.bBoardIdCreatedBy			:= tyBoardAvailableSnd.tyData.sBoardIdCreatedBy <> '';
				tyBoardAvailableSnd.tyAvl.bFailedBoard				:= TRUE;
				tyBoardAvailableSnd.tyAvl.bProductTypeId			:= tyBoardAvailableSnd.tyData.sProductTypeId <> '';
				tyBoardAvailableSnd.tyAvl.bFlippedBoard				:= TRUE;
				tyBoardAvailableSnd.tyAvl.bTopBarcode				:= tyBoardAvailableSnd.tyData.sTopBarcode <> '';
				tyBoardAvailableSnd.tyAvl.bBottomBarcode			:= tyBoardAvailableSnd.tyData.sBottomBarcode <> '';
				tyBoardAvailableSnd.tyAvl.bLength					:= tyBoardAvailableSnd.tyData.rLength <> 0;
				tyBoardAvailableSnd.tyAvl.bWidth					:= (tyBoardAvailableSnd.tyData.rWidth <> 0);
				tyBoardAvailableSnd.tyAvl.bThickness				:= (tyBoardAvailableSnd.tyData.rThickness <> 0);
				tyBoardAvailableSnd.tyAvl.bConveyorSpeed			:= tyBoardAvailableSnd.tyData.rConveyorSpeed <> 0;
				tyBoardAvailableSnd.tyAvl.bTopClearanceHeight		:= (tyBoardAvailableSnd.tyData.rTopClearanceHeight <> 0);
				tyBoardAvailableSnd.tyAvl.bBottomClearanceHeight	:= (tyBoardAvailableSnd.tyData.rBottomClearanceHeight <> 0);
				tyBoardAvailableSnd.tyAvl.bWeight					:= tyBoardAvailableSnd.tyData.rWeight <> 0;
				tyBoardAvailableSnd.tyAvl.bWorkOrderId				:= tyBoardAvailableSnd.tyData.sWorkOrderId <> '';
				tyBoardAvailableSnd.tyAvl.bBatchId			    	:= tyBoardAvailableSnd.tyData.sBatchId <> '';

			ELSE //Take from PCB_In Board Data

				fbParseBrdAvlExternal.p_XMLTable		:= ADR(pa_tyXMLTableDataBrdAvl); //last zone B.A
				fbParseBrdAvlExternal.iTotalIdxWrite	:= p_iXMLTableDataBrdAvlTtlIdx; //last zone
				fbParseBrdAvlExternal;
				tyBoardAvailableSnd	:= fbParseBrdAvlExternal.tyBoardAvailable;
			END_IF

		ELSIF fbSequenceDS.eMsgTypeSnd = HermesMsgTypeRevokeBoardAvl THEN
			fHermesAddOneMsgSend(ADR(a_eMsgSend) , ADR(udiMsgSendBffr) , HermesMsgTypeRevokeBoardAvl);

		ELSIF fbSequenceDS.eMsgTypeSnd = HermesMsgTypeTransportFinished THEN
			fHermesAddOneMsgSend(ADR(a_eMsgSend) , ADR(udiMsgSendBffr) , HermesMsgTypeTransportFinished);

			IF p_bSndCompl = TRUE THEN
				tyTransportFinished.tyData.eTransferState	:= HermesTransferStateComplete;
			ELSIF p_bSndIncompl = TRUE THEN
				tyTransportFinished.tyData.eTransferState	:= HermesTransferStateIncomplete;
			ELSE
				tyTransportFinished.tyData.eTransferState	:= HermesTransferStateNotStarted;
			END_IF
			tyTransportFinished.tyData.sBoardId				:= tyStartTransport.tyData.sBoardId;

			tyTransportFinished.tyAvl.bTransferState		:= TRUE;
			tyTransportFinished.tyAvl.bBoardId				:= TRUE;

		END_IF

	END_IF

END_ACTION
```

#### Act_Background_SequenceTO.st
```iecst
(** 2021-08-01 **)
ACTION Act_Background_SequenceTO:

	IF (eStatus1 <> Error) AND (eStatus2 <> Error) THEN

		//Time Out
		fbSequenceTO.eState				:= fbSequenceDS.eState;
		fbSequenceTO.tConnTimeOut		:= p_tConnTimeOut;
		fbSequenceTO.tTransportTimeOut	:= DINT_TO_TIME(p_diTransferInTO);
		fbSequenceTO(bEn := TRUE);

		IF fbSequenceTO.udiStatus > 0 AND fbSequenceTO.udiStatus < 65534 THEN

			IF fbSequenceTO.udiStatus = 2912 THEN
				eStatus1	:= Error;
				udiStatus1	:= 10106;	//Service Description Interchange Time Out

				fHermesAddOneMsgSend(ADR(a_eMsgSend) , ADR(udiMsgSendBffr) , HermesMsgTypeNotification);

				tyNotificationSnd.tyAvl.bSeverity			:= TRUE;
				tyNotificationSnd.tyAvl.bNotificationCode	:= TRUE;
				tyNotificationSnd.tyAvl.bDescription		:= TRUE;
				tyNotificationSnd.tyData.eSeverity			:= HermesSeverityFatalError;
				tyNotificationSnd.tyData.iNotificationCode	:= UDINT_TO_INT(udiStatus1);
				tyNotificationSnd.tyData.sDescription		:= a_tyAlmText[udiStatus1].sAlmText;

			ELSIF fbSequenceTO.udiStatus = 2913 THEN
				p_bSndIncompl	:= TRUE;

				eStatus2	:= Error;
				udiStatus2	:= 10107;	//Transport Time Out

				fHermesAddOneMsgSend(ADR(a_eMsgSend) , ADR(udiMsgSendBffr) , HermesMsgTypeNotification);

				tyNotificationSnd.tyAvl.bSeverity			:= TRUE;
				tyNotificationSnd.tyAvl.bNotificationCode	:= TRUE;
				tyNotificationSnd.tyAvl.bDescription		:= TRUE;
				tyNotificationSnd.tyData.eSeverity			:= HermesSeverityError;
				tyNotificationSnd.tyData.iNotificationCode	:= UDINT_TO_INT(udiStatus2);
				tyNotificationSnd.tyData.sDescription		:= a_tyAlmText[udiStatus2].sAlmText;

			ELSE
				eStatus2	:= Error;
				udiStatus2	:= fbSequenceTO.udiStatus;

				fHermesAddOneMsgSend(ADR(a_eMsgSend) , ADR(udiMsgSendBffr) , HermesMsgTypeNotification);

				tyNotificationSnd.tyAvl.bSeverity			:= TRUE;
				tyNotificationSnd.tyAvl.bNotificationCode	:= TRUE;
				tyNotificationSnd.tyAvl.bDescription		:= TRUE;
				tyNotificationSnd.tyData.eSeverity			:= HermesSeverityFatalError;
				tyNotificationSnd.tyData.iNotificationCode	:= UDINT_TO_INT(udiStatus2);
				tyNotificationSnd.tyData.sDescription		:= a_tyAlmText[udiStatus2].sAlmText;

			END_IF

		END_IF

	END_IF

END_ACTION
```

#### Act_Background_TCPCloseSvr.st
```iecst
(** 2019-06-10 **)
ACTION Act_Background_TCPCloseSvr:

	//Close Server Connection
	IF p_bInternalUse = FALSE THEN
		fbCloseSvr.udiTCPIdent	:= udiSvrIdent;
		fbCloseSvr(bEn := TRUE);

		IF fbCloseSvr.udiStatus = 0 THEN
			udiSvrIdent		:= 0;
			fbCloseSvr(bEn := FALSE);

		ELSIF fbCloseSvr.udiStatus < 65534 THEN
			udiSvrIdent		:= 0;
			eStatus1		:= Error;

			IF fbCloseSvr.udiStatus = 2300 THEN
				udiStatus1	:= 10146;	//Invalid Ident While Closing TCP
			ELSIF fbCloseSvr.udiStatus = 2310 THEN
				udiStatus1	:= 10147;	//Closing TCP Error
			ELSE
				udiStatus1	:= fbCloseSvr.udiStatus;
			END_IF

		END_IF

	ELSE
		udiSvrIdent	:= 0;

	END_IF

END_ACTION
```

#### Act_Background_TCPSend.st
```iecst
(** 2019-06-10 **)
ACTION Act_Background_TCPSend:

	//Message Send (Generate XML Message)
	IF a_eMsgSend[0] <> HermesMsgTypeNA THEN

		IF a_eMsgSend[0] = HermesMsgTypeCheckAlive THEN
			fHermesFormCheckAlive(ADR(a_tyXMLTableDataSnd) , p_tyDTStructure , tyCheckAliveSnd);
			fTableConvertToXML(ADR(sSnd) , ADR(udiSndMsgLen) , SIZEOF(sSnd) , ADR(a_tyXMLTableDataSnd) , ADR(a_tyXMLTableDataSnd[0].sTitle) , ADR(a_tyXMLTableDataSnd[0].sValue) , ADR(a_tyXMLTableDataSnd[0].uiSize) , SIZEOF(a_tyXMLTableDataSnd[0]) , 12);

		ELSIF a_eMsgSend[0] = HermesMsgTypeCheckAlivePing THEN
			fHermesFormCheckAlive(ADR(a_tyXMLTableDataSnd) , p_tyDTStructure , tyCheckAlivePingSnd);
			fTableConvertToXML(ADR(sSnd) , ADR(udiSndMsgLen) , SIZEOF(sSnd) , ADR(a_tyXMLTableDataSnd) , ADR(a_tyXMLTableDataSnd[0].sTitle) , ADR(a_tyXMLTableDataSnd[0].sValue) , ADR(a_tyXMLTableDataSnd[0].uiSize) , SIZEOF(a_tyXMLTableDataSnd[0]) , 12);

		ELSIF a_eMsgSend[0] = HermesMsgTypeCheckAlivePong THEN
			fHermesFormCheckAlive(ADR(a_tyXMLTableDataSnd) , p_tyDTStructure , tyCheckAlivePongSnd);
			fTableConvertToXML(ADR(sSnd) , ADR(udiSndMsgLen) , SIZEOF(sSnd) , ADR(a_tyXMLTableDataSnd) , ADR(a_tyXMLTableDataSnd[0].sTitle) , ADR(a_tyXMLTableDataSnd[0].sValue) , ADR(a_tyXMLTableDataSnd[0].uiSize) , SIZEOF(a_tyXMLTableDataSnd[0]) , 12);

		ELSIF a_eMsgSend[0] = HermesMsgTypeServiceDescription THEN
			fHermesFormServiceDescription(ADR(a_tyXMLTableDataSnd) , p_tyDTStructure , tyServiceDescriptionSnd);
			fTableConvertToXML(ADR(sSnd) , ADR(udiSndMsgLen) , SIZEOF(sSnd) , ADR(a_tyXMLTableDataSnd) , ADR(a_tyXMLTableDataSnd[0].sTitle) , ADR(a_tyXMLTableDataSnd[0].sValue) , ADR(a_tyXMLTableDataSnd[0].uiSize) , SIZEOF(a_tyXMLTableDataSnd[0]) , 30);

		ELSIF a_eMsgSend[0] = HermesMsgTypeNotification THEN
			fHermesFormNotification(ADR(a_tyXMLTableDataSnd) , p_tyDTStructure , tyNotificationSnd);
			fTableConvertToXML(ADR(sSnd) , ADR(udiSndMsgLen) , SIZEOF(sSnd) , ADR(a_tyXMLTableDataSnd) , ADR(a_tyXMLTableDataSnd[0].sTitle) , ADR(a_tyXMLTableDataSnd[0].sValue) , ADR(a_tyXMLTableDataSnd[0].uiSize) , SIZEOF(a_tyXMLTableDataSnd[0]) , 14);

		ELSIF a_eMsgSend[0] = HermesMsgTypeBoardAvailable THEN
			fHermesFormBoardAvailable(ADR(a_tyXMLTableDataSnd) , p_tyDTStructure , tyBoardAvailableSnd);
			fTableConvertToXML(ADR(sSnd) , ADR(udiSndMsgLen) , SIZEOF(sSnd) , ADR(a_tyXMLTableDataSnd) , ADR(a_tyXMLTableDataSnd[0].sTitle) , ADR(a_tyXMLTableDataSnd[0].sValue) , ADR(a_tyXMLTableDataSnd[0].uiSize) , SIZEOF(a_tyXMLTableDataSnd[0]) , 88);//50

		ELSIF a_eMsgSend[0] = HermesMsgTypeRevokeBoardAvl THEN
			fHermesFormRevokeBoardAvailable(ADR(a_tyXMLTableDataSnd) , p_tyDTStructure);
			fTableConvertToXML(ADR(sSnd) , ADR(udiSndMsgLen) , SIZEOF(sSnd) , ADR(a_tyXMLTableDataSnd) , ADR(a_tyXMLTableDataSnd[0].sTitle) , ADR(a_tyXMLTableDataSnd[0].sValue) , ADR(a_tyXMLTableDataSnd[0].uiSize) , SIZEOF(a_tyXMLTableDataSnd[0]) , 8);

		ELSIF a_eMsgSend[0] = HermesMsgTypeMachineReady THEN
			eStatus1	:= Error;
			udiStatus1	:= 10135;	//Machine Ready Request To Send From Upstream Hermes

		ELSIF a_eMsgSend[0] = HermesMsgTypeRevokeMachineReady THEN
			eStatus1	:= Error;
			udiStatus1	:= 10136;	//Revoke Machine Ready Request To Send From Upstream Hermes

		ELSIF a_eMsgSend[0] = HermesMsgTypeStartTransport THEN
			eStatus1	:= Error;
			udiStatus1	:= 10137;	//Start Transport Request To Send From Upstream Hermes

		ELSIF a_eMsgSend[0] = HermesMsgTypeStopTransport THEN
			eStatus1	:= Error;
			udiStatus1	:= 10110;	//Stop Transport Request To Send From Upstream Hermes

		ELSIF a_eMsgSend[0] = HermesMsgTypeTransportFinished THEN
			fHermesFormTransportFinished(ADR(a_tyXMLTableDataSnd) , p_tyDTStructure , tyTransportFinished);
			fTableConvertToXML(ADR(sSnd) , ADR(udiSndMsgLen) , SIZEOF(sSnd) , ADR(a_tyXMLTableDataSnd) , ADR(a_tyXMLTableDataSnd[0].sTitle) , ADR(a_tyXMLTableDataSnd[0].sValue) , ADR(a_tyXMLTableDataSnd[0].uiSize) , SIZEOF(a_tyXMLTableDataSnd[0]) , 12);

		ELSIF a_eMsgSend[0] = HermesMsgTypeSetConfiguration THEN
			eStatus1	:= Error;
			udiStatus1	:= 10138;	//Set Configuration Request To Send From Upstream Hermes

		ELSIF a_eMsgSend[0] = HermesMsgTypeGetConfiguration THEN
			eStatus1	:= Error;
			udiStatus1	:= 10139;	//Get Configuration Request To Send From Upstream Hermes

		ELSIF a_eMsgSend[0] = HermesMsgTypeCurrConfiguration THEN
			eStatus1	:= Error;
			udiStatus1	:= 10140;	//Current Configuration Request To Send From Upstream Hermes

		ELSIF a_eMsgSend[0] = HermesMsgTypeBoardForecast THEN
			fHermesFormBoardForecast(ADR(a_tyXMLTableDataSnd) , p_tyDTStructure , tyBoardForecastSnd);
			fTableConvertToXML(ADR(sSnd) , ADR(udiSndMsgLen) , SIZEOF(sSnd) , ADR(a_tyXMLTableDataSnd) , ADR(a_tyXMLTableDataSnd[0].sTitle) , ADR(a_tyXMLTableDataSnd[0].sValue) , ADR(a_tyXMLTableDataSnd[0].uiSize) , SIZEOF(a_tyXMLTableDataSnd[0]) , 50);

		ELSIF a_eMsgSend[0] = HermesMsgTypeQueryBoardInfo THEN
			eStatus1	:= Error;
			udiStatus1	:= 10142;	//Query Board Info Request To Send From Upstream Hermes

		ELSIF a_eMsgSend[0] = HermesMsgTypeSendBoardInfo THEN
			fHermesFormSendBoardInfo(ADR(a_tyXMLTableDataSnd) , p_tyDTStructure , tySendBoardInfo);
			fTableConvertToXML(ADR(sSnd) , ADR(udiSndMsgLen) , SIZEOF(sSnd) , ADR(a_tyXMLTableDataSnd) , ADR(a_tyXMLTableDataSnd[0].sTitle) , ADR(a_tyXMLTableDataSnd[0].sValue) , ADR(a_tyXMLTableDataSnd[0].uiSize) , SIZEOF(a_tyXMLTableDataSnd[0]) , 34);

		ELSIF a_eMsgSend[0] = HermesMsgTypeCommand THEN
			fHermesFormCommand(ADR(a_tyXMLTableDataSnd) , p_tyDTStructure , tyCommandSnd);
			fTableConvertToXML(ADR(sSnd) , ADR(udiSndMsgLen) , SIZEOF(sSnd) , ADR(a_tyXMLTableDataSnd) , ADR(a_tyXMLTableDataSnd[0].sTitle) , ADR(a_tyXMLTableDataSnd[0].sValue) , ADR(a_tyXMLTableDataSnd[0].uiSize) , SIZEOF(a_tyXMLTableDataSnd[0]) , 10);

		END_IF

		//Message Send
		IF p_bInternalUse = FALSE THEN
			fbSend.udiTCPIdent	:= udiClntIdent;
			fbSend.udiSndSize	:= udiSndMsgLen;
			fbSend(bEn := TRUE);
		ELSE
			sInternalSnd	:= sSnd;
		END_IF

		IF (fbSend.udiStatus = 0) OR (p_bInternalUse = TRUE) THEN

			fLogDTConvert(ADR(sDT) , p_dtCurrDT);
			memset(ADR(a_sLogList[udiLogCntr]) , 0 , SIZEOF(a_sLogList[udiLogCntr]));
			memcpy(ADR(a_sLogList[udiLogCntr]) + LEN(a_sLogList[udiLogCntr]) , ADR(sDT) , LEN(sDT));
			memcpy(ADR(a_sLogList[udiLogCntr]) + LEN(a_sLogList[udiLogCntr]) , ADR('$r$n') , LEN('$r$n'));
			memcpy(ADR(a_sLogList[udiLogCntr]) + LEN(a_sLogList[udiLogCntr]) , ADR('SND_TO_DS$r$n') , LEN('SND_TO_DS$r$n'));
			memcpy(ADR(a_sLogList[udiLogCntr]) + LEN(a_sLogList[udiLogCntr]) , ADR(sSnd) , LEN(sSnd));
			memcpy(ADR(a_sLogList[udiLogCntr]) + LEN(a_sLogList[udiLogCntr]) , ADR('$r$n$r$n') , LEN('$r$n$r$n'));

			udiLogCntr	:= udiLogCntr + 1;
			IF udiLogCntr = 11 THEN
				udiLogCntr	:= 1;
			END_IF

			Act_Background_NotificationSnd;
			fHermesRmvOneMsgSend(ADR(a_eMsgSend) , ADR(udiMsgSendBffr));

			fbSend(bEn := FALSE);

		ELSIF (fbSend.udiStatus = 2321) AND (p_bInternalUse = FALSE) THEN
			bRstConnection	:= TRUE;

		ELSIF (fbSend.udiStatus < 65534) AND (p_bInternalUse = FALSE) THEN
			eStatus1	:= Error;

			IF fbSend.udiStatus = 2300 THEN
				udiStatus1	:= 10143;	//Invalid Ident While Sending Data
			ELSIF fbSend.udiStatus = 2320 THEN
				udiStatus1	:= 10144;	//TCP Retry Send Data Error While Sending Data
			ELSIF fbSend.udiStatus = 2322 THEN
				udiStatus1	:= 10145;	//TCP Send Data Error
			ELSE
				udiStatus1	:= fbSend.udiStatus;
			END_IF

		END_IF

	END_IF

END_ACTION
```

#### Act_InitGlobal.st
```iecst
(** 2019-05-04 **)
ACTION Act_InitGlobal:

	(* Always Change If Project Change *)

	//Pass Data To Link
	p_bLinkStartupRun ACCESS p_StartupRun;
	p_eLinkMcParamDSCommMod ACCESS p_McParamDSComm2Mod;

	p_eLinkConvDir ACCESS p_NtParamProjConvDir;
	p_bLinkConvGdBrd ACCESS p_ConvGdBrd;
	p_bLinkDILeftSen ACCESS p_DIConvLftSen;
	p_bLinkDIRightSen ACCESS p_DIConvRgtSen;
	p_bLinkConvHvBrd ACCESS p_OpsInvertHvBrd;
	//Pass Data To Internal Use
	p_udiRstErr ACCESS p_RstErrReset;
	p_bPrep ACCESS p_NtParamHermesPrep;
	p_tyParam ACCESS p_HermesDSParam2;
	p_sIPAddr ACCESS p_HWInfoIPAddr;
	pa_usiMacAddr ACCESS p_HWInfoMacAddr;
	p_tyDTStructure ACCESS p_TimeCurrDTStruct;
	p_dtCurrDT ACCESS p_TimeCurrDT;
	p_sMcId ACCESS p_McParamMcNm;
	p_sRecipeNm ACCESS p_ProdRcpCurrRcp0Nm;
	p_sRecipeZone1Nm ACCESS p_ProdRcpCurrRcp1Nm;
	//p_sWorkOrderId ACCESS p_SvyHermesWorkOrderId; //Work Order Id from SupervisoryHermes
	//p_sBatchId ACCESS p_SvyHermesBatchId; //Batch Id from SupervisoryHermes
	p_diWidthInUM ACCESS p_ProdRcpCurrRcp0Width;
	p_diWidthZone1InUM ACCESS p_ProdRcpCurrRcp1Width;
	p_udiAliveIdleTimeInSec ACCESS p_NtParamDSHermes2AliveTmInSec;
	p_tConnTimeOut ACCESS p_NtParamDSHermes2ConnTO;
	p_diTransferInTO ACCESS p_McParamTranOutErrDlyTm;
	pa_tyXMLTableDataBrdAvl ACCESS p_HermesBrdAvlDataTableLastZ;
	p_iXMLTableDataBrdAvlTtlIdx ACCESS p_HermesBrdAvlDataTtlIdxLastZ;
	p_bNewBrdAvlFirstZone ACCESS p_HermesBrdAvlDataNewBrdAvl1stZ;
	p_bNewBrdAvlLastZone ACCESS p_HermesBrdAvlDataNewBrdAvlLastZ;
	p_bOpsRun ACCESS p_OpsRun;
	p_bInterruptSen ACCESS p_DIConvRgtSen;
	p_udiFileKeepDay ACCESS p_NtParamDSHermes2FileKeepDay;
	p_sRetainFileName ACCESS p_NtParamDSHermesRetainFileNm;
	p_sProgNm ACCESS p_NtParamDSHermes2ProgNm;
	p_bNtSettingsLoadDone ACCESS p_StartupNtSettingsLoadDone;
	p_sRmtMcId ACCESS p_RmtHermesCurrentConfMcId;
	p_bRmtPrep ACCESS p_NtParamHermesRmtPrep;
	p_bRmtEn ACCESS p_McParamHermesRmtEn;

	p_bUSHermesStopTransport ACCESS p_USHermesStopTransportSnd;

	p_tyUSHermestyBoardAvailable ACCESS p_USHermestyBoardAvailable;
	p_bNtParamProjInvertOncePrep ACCESS p_NtParamProjInvertOncePrep;
	p_bNtParamProjInvertTwicePrep ACCESS p_NtParamProjInvertTwicePrep;

	//for reverse condition
	//p_bUSHermesReverseDSSendBFId ACCESS p_USHermesReverseDSSendBFId;
	//p_bUSHermesProcessRouteTrigger ACCESS p_USHermesProcessRouteTrigger;
	p_usiUSHermesReverseDSSendBFId ACCESS p_HermesReverseDS2SendBFId;
	p_bUSHermesProcessRouteTrigger ACCESS p_USHermesProcessRouteTrigger;
	pa_RevtyXMLTableDataBrdAvl  ACCESS p_USHermesTableDataBrdAvl;
	p_ReviXMLTableDataBrdAvlTtlIdx ACCESS  p_USHermesTableDataBrdAvlTtlIdx;

	//BoardForecast
	p_tyUSBoardArrivedData  ACCESS p_USHermesBoardArrivedData;
	//Board Available

	p_bRcvBoardInfo ACCESS p_USHermesRcvBoardInfoOk;
	p_tyBoardInfoData ACCESS p_USHermesBoardInfoData;

	p_bConvInitDone ACCESS p_OpsInvertStepInitConv;

	p_bHermesSwitchtoRvrseTransport ACCESS p_HermesSwitchtoReverseTransport;
	(* Always Change If Project Change *)

END_ACTION
```

#### Act_Initial.st
```iecst
(** 2021-08-01 **)
ACTION Act_Initial:

	//Initial
	sStatTxt	:= a_sStatText[eStat];

	fbCreateSvr.udiSndBffrSize		:= p_udiSndBffrSize;
	fbCreateSvr.udiRcvBffrSize		:= p_udiRcvBffrSize;
	fbCreateSvr.udiAliveIdleTmInSec	:= p_udiAliveIdleTimeInSec;
	fbCreateSvr(bEn := FALSE);

	fbListen(bEn := FALSE);

	fbRcv.udiBffrSize	:= SIZEOF(sRcv);
	fbRcv.p_BffrDest	:= ADR(sRcv);
	fbRcv(bEn := FALSE);

	fbSend.p_BffrDest	:= ADR(sSnd);
	fbSend(bEn := FALSE);

	fbCloseSvr(bEn := FALSE);
	fbCloseClnt(bEn := FALSE);

	fbParseXMLTable.p_XMLTable	:= ADR(a_tyXMLTableDataRcv);

	fbCheckAlive(bEn := FALSE);

	fbCheckAliveSendPing(bEn := FALSE);

	fbCheckAliveRcvPing(bEn := FALSE);

	fbSequenceDS.p_tyMsgTypeRcv	:= ADR(tyMsgTypeRcv);
	fbSequenceDS(bEn := FALSE);

	fbSequenceTO(bEn := FALSE);

	fbFileAppend1.sDevice	:= 'Log';
	fbFileAppend1(bEn := FALSE);

	fbFileOldDel1.sDevice			:= 'Log';
	fbFileOldDel1.sPath				:= '';
	fbFileOldDel1.sKeyword			:= p_sProgNm;
	fbFileOldDel1.udiFileKeepDay	:= p_udiFileKeepDay;
	fbFileOldDel1(bEn := FALSE);

	fbFileRead1.sDevice			:= 'Retain';
	fbFileRead1.sFile			:= p_sRetainFileName;
	fbFileRead1.udiOffset		:= 0;
	fbFileRead1.p_Dest			:= ADR(a_tyBoardDepartedInfo);
	fbFileRead1.udiLen			:= SIZEOF(a_tyBoardDepartedInfo);
	fbFileRead1(bEn := FALSE);

	fbFileWrite1.sDevice		:= 'Retain';
	fbFileWrite1.sFile			:= p_sRetainFileName;
	fbFileWrite1.udiOffset		:= 0;
	fbFileWrite1.udiOption		:= 0;
	fbFileWrite1.p_Src			:= ADR(a_tyBoardDepartedInfoWr);
	fbFileWrite1.udiLen			:= SIZEOF(a_tyBoardDepartedInfoWr);
	fbFileWrite1(bEn := FALSE);

END_ACTION
```

#### Act_Link.st
```iecst
(** 2019-04-08 **)
ACTION Act_Link:

	//Receive Alive Time
	p_tyParam.tRcvAlive	:= p_tyParam.tSndAlive * 2;

	//Ready Send //need to uncomment back
	p_bRdySnd ACCESS p_OpsInvertStepDSCommTmr;

	//boardforecast
	bNewProduct := EDGEPOS(p_sRecipeNm <> p_sRecipeZone1Nm) AND p_bLinkStartupRun = FALSE;
	bNewWidth := EDGEPOS(p_diWidthInUM <> p_diWidthZone1InUM) AND p_bLinkStartupRun = FALSE;
	bAllZoneEmpty := p_bLinkDIRightSen = FALSE AND p_bLinkDILeftSen = FALSE AND p_bLinkConvHvBrd = FALSE;

	//Transfer Finished
	IF NOT(p_bHermesSwitchtoRvrseTransport) THEN //(p_eLinkConvDir = ConvDirLToR) OR (p_eLinkConvDir = ConvDirRToR) THEN
		IF EDGENEG(p_bLinkDIRightSen) THEN
			p_bSndCompl	:= TRUE;
		END_IF
		bFirstZoneHaveBoard :=  p_bLinkDILeftSen= TRUE;
		bFirstZoneEndSen :=  p_bLinkDIRightSen = FALSE;
	ELSE
		IF EDGENEG(p_bLinkDILeftSen) THEN
			p_bSndCompl	:= TRUE;
		END_IF
		bFirstZoneHaveBoard := p_bLinkDIRightSen = TRUE;
		bFirstZoneEndSen :=  p_bLinkDILeftSen= FALSE;
	END_IF

	//Good Bad Board
	IF p_bLinkConvGdBrd = TRUE THEN
		p_eFailedBoard	:= HermesGoodBoard;
	ELSE
		p_eFailedBoard	:= HermesFailedBoard;
	END_IF

	//Flip Board
//	IF p_tyUSHermestyBoardAvailable.tyData.eFlippedBoard = 2 THEN
//		p_eFlippedBoard := 1;
//
//	ELSIF p_tyUSHermestyBoardAvailable.tyData.eFlippedBoard = 1 THEN
//		p_eFlippedBoard := 2;
//
//	ELSE
//		p_eFlippedBoard := 0;
//	END_IF

	//first zone have board
	//Machine First Zone have board
	//p_bFirstZoneHaveBoard := (p_bUSHermesStopTransport AND p_bOpsGConvHvBrd) OR (p_bOpsGConvHvBrd AND p_bUSHermesTransporting = FALSE); //Zone 1 have board, either PCB_In from upstream Or Manually load PCB at Zone 1

END_ACTION
```
